// TwinCAT 3 PLC project Steamer
// ProgramVersion: 3.1.4026.25
// libraries:
//   Tc2_Standard, * (Beckhoff Automation GmbH)
//   Tc2_System, * (Beckhoff Automation GmbH)
//   Tc2_Utilities, * (Beckhoff Automation GmbH)
// project tree:
//   DUTs/Enumerations/ E_FaultId.TcDUT, E_HmiMessage.TcDUT (not stored), E_SystemState.TcDUT, E_WaterFillMode.TcDUT (not stored)
//   DUTs/Structures/ ST_Faults.TcDUT, ST_HmiCommand.TcDUT, ST_HmiSetpoints.TcDUT, ST_HmiStatus.TcDUT, ST_ProcessValues.TcDUT
//   GVLs/ GVL_HMI.TcGVL, GVL_IO.TcGVL, GVL_SysParameters.TcGVL
//   / PlcTask.TcTTO
//   POUs/ FB_FaultMonitor.TcPOU, FB_Hmi.TcPOU, FB_ProcessCalcs.TcPOU, FB_OutputHandler.TcPOU, FB_PressureControl.TcPOU, FB_Purge.TcPOU, FB_SpaFlush.TcPOU, FB_StateMachine.TcPOU, FB_WaterFill.TcPOU, MAIN.TcPOU
// real-time tasks:
//   TASK PlcTask: cycle T#10ms, priority 20, ADS port 350
// I/O:
//   DEVICE Device 1 (EtherCAT), AmsNetId 5.177.96.78.2.1
//     Term 1 (EK1200) [EK1200-7000 EtherCAT Power supply (1,5A E-Bus)]
//       Term 2 (EL1008) [EL1008 8Ch. Dig. Input 24V, 3ms]
//       Term 3 (EL2008) [EL2008 8Ch. Dig. Output 24V, 0.5A]
//       Term 4 (EL2008) [EL2008 8Ch. Dig. Output 24V, 0.5A]
//       Term 11 (EL3052) [EL3052 2Ch. Ana. Input 4-20mA]
//       Term 5 (EL3314) [EL3314 4Ch. Ana. Input Thermocouple (TC)]
//       Term 13 (EL6652-0010) [EL6652-0010 EtherNet/IP Adapter (Slave)]
//       Term 6 (EL9011) [EL9011 End Terminal]
// variable links:
//   Steamer/Steamer Instance <-> Device 1 (EtherCAT)/Term 1 (EK1200)/Term 11 (EL3052)
//     PlcTask Inputs/GVL_IO.aiPT1_UpstreamPressure <-> AI Standard Channel 1/Value
//     PlcTask Inputs/GVL_IO.aiPT2_DownstreamPressure <-> AI Standard Channel 2/Value
//   Steamer/Steamer Instance <-> Device 1 (EtherCAT)/Term 1 (EK1200)/Term 2 (EL1008)
//     PlcTask Inputs/GVL_IO.biLS1_WaterMidLevel <-> Channel 3/Input
//     PlcTask Inputs/GVL_IO.biLS2_WaterHighLevel <-> Channel 4/Input
//     PlcTask Inputs/GVL_IO.biLS3_WaterLowLevel <-> Channel 5/Input
//     PlcTask Inputs/GVL_IO.biTankFloodFault <-> Channel 2/Input
//   Steamer/Steamer Instance <-> Device 1 (EtherCAT)/Term 1 (EK1200)/Term 3 (EL2008)
//     PlcTask Outputs/GVL_IO.boH1_UpstreamHeater <-> Channel 5/Output
//     PlcTask Outputs/GVL_IO.boH2_SpaHeater <-> Channel 6/Output
//     PlcTask Outputs/GVL_IO.boH3_FlowmeterHeater <-> Channel 7/Output
//     PlcTask Outputs/GVL_IO.boH4_ExternalHeater <-> Channel 8/Output
//     PlcTask Outputs/GVL_IO.boSV1_DrainValve <-> Channel 1/Output
//     PlcTask Outputs/GVL_IO.boSV2_SpaValve <-> Channel 2/Output
//     PlcTask Outputs/GVL_IO.boSV3_DeliveryValve <-> Channel 3/Output
//     PlcTask Outputs/GVL_IO.boSV4_WaterInletValve <-> Channel 4/Output
//   Steamer/Steamer Instance <-> Device 1 (EtherCAT)/Term 1 (EK1200)/Term 5 (EL3314)
//     PlcTask Inputs/GVL_IO.aiTC1_SpaTemp <-> TC Inputs Channel 1/Value
//     PlcTask Inputs/GVL_IO.aiTC2_FlometerTemp <-> TC Inputs Channel 2/Value
//     PlcTask Inputs/GVL_IO.aiTC3_ExternalTemp <-> TC Inputs Channel 3/Value
//     PlcTask Inputs/GVL_IO.aiTC4_DeliveryTemp <-> TC Inputs Channel 4/Value

CONFIGURATION Steamer
    RESOURCE PLC ON TwinCAT3
        TASK PlcTask(INTERVAL := T#10ms, PRIORITY := 20);
        PROGRAM MAIN WITH PlcTask : MAIN;
    END_RESOURCE
END_CONFIGURATION

// ---- DUTs/Enumerations/E_FaultId.TcDUT
//=============================================================================
// E_FaultId
//-----------------------------------------------------------------------------
// Identifies WHICH fault tripped first. FB_FaultMonitor latches one of these
// on the transition from healthy to faulted and holds it until ResetAll().
//
// The numeric values are the legacy HMI message-table indices, so the existing
// message strings on the panel keep working without a translation layer.
// Where the legacy reused one index for several distinct causes, the causes
// are split into separate IDs here and the duplicated index is noted.
//=============================================================================
{attribute 'qualified_only'}
{attribute 'strict'}
{attribute 'to_string'}
TYPE E_FaultId :
(
    None                    := 0,

    // --- hardware / utilities -------------------------------------------
    PowerFault              := 1,
	CabinetFlood            := 2,
    PneumaticLow            := 3,

    // --- pressure -------------------------------------------------------
    UpstreamOverPress       := 11,
    DownstreamOverPress     := 12,
    DownstreamStartHigh     := 13,
    StartupDiffPressTimeout := 14,
    Pt1Hardware             := 15,
    Pt2Hardware             := 16,

    // Transducer cross-check failure. Legacy shared index 58 with the
    // timeout above; split so first-out can tell them apart. Point the HMI
    // message table at 58 if a distinct string is not wanted.
    StartupDiffPressXCheck  := 17,

    // --- water ----------------------------------------------------------
    WaterFill               := 21,
    WaterRegulation         := 22,
    WaterEmpty              := 23,
	WaterOverFill			:= 24,
    VesselPurgeTimeout      := 25,

    // --- temperature: over-limit ----------------------------------------
    SpaOverTemp             := 31,
    FlowMeterOverTemp       := 32,
    ExternalOverTemp        := 33,
    DownstreamOverTemp      := 34,

    // --- temperature: warm-up failures ----------------------------------
    SpaWarmupTimeout        := 41,
    FlowMeterWarmupTimeout  := 42,
    ExternalWarmupTimeout   := 43,
    DownstreamWarmupTimeout := 44,

    // Legacy reused index 76 for all three external-line faults. Split so
    // the operator can tell "TC not bonded to heater" from "line went cold".
    ExternalNoTempRise      := 51,
    ExternalLowAtReady      := 52,

    // --- flow -----------------------------------------------------------
    FlowRateError           := 61,

    // --- new in this system ---------------------------------------------
    HmiCommLoss             := 300
) INT;
END_TYPE

// ---- DUTs/Enumerations/E_SystemState.TcDUT
{attribute 'qualified_only'}
{attribute 'strict'}
{attribute 'to_string'}
TYPE E_SystemState :
(
    // --- Boot / idle ---------------------------------------------------
    InitController      := 0, 	// Controller Initialization (one-shot config, params, PID setup)
    SesOff              := 70,  // SES Off (idle / standby, waiting for SES ON command)

    // --- Startup sequence ----------------------------------------------
    CheckIfHot          := 10,  // Check if system was just running (hot restart shortcut)
    FillWater       	:= 20,  // SES Initialization - Fill Water
    PurgeVessel     	:= 30,  // SES Initialization - Purge Vessel
    SetDiffPressure 	:= 40,  // SES Initialization - Setting Differential Pressure
    InitMain       		:= 50,  // SES Initialization - Main (final checks before flow)

    // --- Run -------------------------------------------------------------
    SteamFlowing        := 60,  // Steam Flowing (normal production, PID flow control)

    // --- Service / abnormal ----------------------------------------------
    Maintenance         := 80,  // Maintenance mode (manual actuation, loopback)
    Fault               := 99   // Fault (latched; operator reset returns to InitController)
	
) INT;
END_TYPE

// ---- DUTs/Structures/ST_Faults.TcDUT
//=============================================================================
// ST_Faults
//-----------------------------------------------------------------------------
// One named BOOL per fault, replacing the legacy B1600.x / B1601.x / B1602.x
// bit-of-word addressing. Names taken from the element documentation table
// in the DS6 source. Legacy address noted per field for commissioning.
// pack_mode 1: each BOOL = 1 byte, so pyads can map this with a simple
// structure_def or read it as a byte array.
//=============================================================================
{attribute 'pack_mode' := '1'}
TYPE ST_Faults :
STRUCT
	// --- Legacy system faults --------------------------------------------
    bAnyFault					: BOOL;   	// High when any fault is active
    bPowerFault          		: BOOL;   	// Power fault input high
	bCabinetFlood        		: BOOL;   	// Cabinet flood fault
    bPneumaticLow        		: BOOL;   	// Pneumatic air pressure low
    bUpstreamOverPress   		: BOOL;   	// Upstream over pressure
    bDownstreamOverPress 		: BOOL;   	// Downstream over pressure
    bPt1HardwareFault      		: BOOL;   	// PT1 hardware fault
    bPt2HardwareFault      		: BOOL;   	// PT2 hardware fault
	bSpaOverTemp				: BOOL;		// SPA greater than max temp stpt
	bFlowmeterOverTemp			: BOOL;		// fm greater then max temp stpt
	bExtOverTemp				: BOOL;		// external temp greater than max stpt
	bDownstreamOverTemp			: BOOL;		// delivery temp greater than max stpt
	bSpaWarmupTimeout			: BOOL;		// spa temp below stpt after timeout
	bFlowmeterWarmupTimeout		: BOOL;		// fm temp below stpt after timeout
	bExtWarmupTimeout			: BOOL;		// external temp below stpt after timeout
	bDownstreamWarmupTimeout	: BOOL;		// ds temp below stpt after timeout
	bExtTempDecoupled			: BOOL;		// external temp disconnected from heater
	bExtTempLow					: BOOL;		// external temp low after steam ready
    bWaterEmpty          		: BOOL; 	// empty water level fault
	bWaterOverFill				: BOOL;		// water too full fault
	bWaterFillTimeout          	: BOOL; 	// water not full after timeout 
	bWaterDrainTimeout          : BOOL; 	// water not empty after timeout
	bWaterRegulationFault		: BOOL;		// water PID stuck on too long
	bPurgeTimeout				: BOOL;		// vessel purge incomplete after timeout
	bDownstreamStartOverPress	: BOOL;		// vessel not properly vented before restart
	bStartDpTimeout				: BOOL;		// diff pressure timeout before reaching stpt
	bStartDpHardwareFault		: BOOL;		// pressure outside of allowable variance
	bFlowFault					: BOOL;		// flow to dp ratio exceeds calibrated max

    // --- New-system faults ---------------------------------------
    bHmiCommLoss         : BOOL;   // (new) RPi heartbeat timeout
	
END_STRUCT
END_TYPE

// ---- DUTs/Structures/ST_HmiCommand.TcDUT
//=============================================================================
// ST_HmiCommand
//-----------------------------------------------------------------------------
// Direction: Pi -> PLC. Consume-on-read pattern:
//   * Pi writes TRUE to a command bit (pyads write_by_name).
//   * FB_Hmi latches it into its outputs for exactly one PLC cycle,
//     then writes FALSE back. The Pi never needs to clear anything.
//
//=============================================================================
{attribute 'pack_mode' := '1'}
TYPE ST_HmiCommand :
STRUCT
	// --- Heartbeat -------------------------------------------------------------
    nHmiHeartbeat   : UDINT;   // Pi increments each poll cycle; never reset

    // --- Run page buttons ---------------------------------------------------
    bSesOn          	: BOOL;    // start command
    bSesOff         	: BOOL;    // stop command 
	bSteamDeliveryOn	: BOOL;    // steam delivery enable
	bSteamDeliveryOff	: BOOL;    // steam delivery disable

    // --- Alarms page --------------------------------------------------------
    bFaultReset     	: BOOL;    // reset all faults
    bFaultAck       	: BOOL;    // acknowledge (silences banner, faults stay listed)

    // --- Maintenance page ---------------------------------------------------
    bEnterMaint     	: BOOL;    				// request Maintenance state
    bExitMaint      	: BOOL;    				// leave Maintenance 
    aValveCmd      		: ARRAY[1..4] OF BOOL;  // SV1 drain, SV2 main, SV3 process, SV4 water
    bDrainMode      	: BOOL;    				// drain mode
	bDpControlOn   		: BOOL;    				// suspend diff pressure control
    bDpControlOff   	: BOOL;    				// suspend diff pressure control
	bTempControlOn	 	: BOOL;    				// suspend purifier temp control
    bTempControlOff 	: BOOL;    				// suspend purifier temp control
    bExtHeaterOn		: BOOL;    				// external heater enable
	bExtHeaterOff		: BOOL;					// extermal heater disable	
	bAutofillOn			: BOOL;					// toggle autofill enable when running
	bAutofillOff		: BOOL;					// toggle autofill off

    // --- Config page --------------------------------------------------------
    bApplySetpoints : BOOL;    // pulse: validate + apply stSetpointRequest

END_STRUCT
END_TYPE

// ---- DUTs/Structures/ST_HmiSetpoints.TcDUT
//=============================================================================
// ST_HmiSetpoints
//-----------------------------------------------------------------------------
// Direction: Pi -> PLC (request) and PLC -> Pi (applied echo in ST_HmiStatus).
// Pi writes the whole struct, then pulses stCommand.bApplySetpoints.
// FB_Hmi clamps each value to ST_SetpointLimits before applying, and the
// clamped result is echoed in ST_HmiStatus.rSet*Applied so the UI always
// shows the truth, not the request.
//=============================================================================
{attribute 'pack_mode' := '1'}
TYPE ST_HmiSetpoints :
STRUCT
	bSetPurgeOnStartup	: BOOL := FALSE;	// 
	rSetFlow       		: REAL;  			// requested flow setpoint      [SLM]
    //rSetDsPressure 		: REAL; 			// downstream pressure setpoint [Torr]
	rSetElevation		: REAL;				// meters above seal level [MASL] 
	bSetSize25L			: BOOL;				// set size to 25L, FALSE = 50L
	sSetEipAddress		: STRING(15);		// string to represent EthernetIP address
END_STRUCT
END_TYPE

// ---- DUTs/Structures/ST_HmiStatus.TcDUT
//=============================================================================
// ST_HmiStatus
//-----------------------------------------------------------------------------
// EVERYTHING the RPi HMI displays, packed into ONE struct so pyads can
// refresh the whole UI with a single read:
//     plc.read_by_name('GVL_HMI.stStatus', structure_def=ST_HMI_STATUS)
//
// Direction: PLC -> Pi only. The Pi must never write this struct.
// pack_mode 1: byte-aligned, no padding — pyads structure_def matches 1:1.
//=============================================================================
{attribute 'pack_mode' := '1'}
TYPE ST_HmiStatus :
STRUCT
    // --- Liveness / handshake -------------------------------------------
    nPlcHeartbeat    	: UDINT;             	// increments every PLC cycle group; Pi checks it changes
    nHmiHeartbeatEcho 	: UDINT;           		// last heartbeat value received from Pi (debug aid)
    bHmiOnline      	: BOOL;              	// PLC's view: Pi heartbeat is alive

    // --- System state ----------------------------------------------------
    eState          	: E_SystemState;     	// current state (INT under the hood)
    sStateName      	: STRING(31);        	// human-readable, e.g. 'SteamFlowing' (state pill)
    bReady          	: BOOL;              	// green Ready dot (temps in band, no faults)
    bAlarmActive    	: BOOL;              	// red Alarm dot (any fault bit set)
    nActiveFaults   	: UINT;              	// count of active fault bits (Alarms page stat card)

    // --- Process data ------------------------------------------------------
    stProcess       	: ST_ProcessValues;  	// pressures, temps, flow, water level
	bFillComplete		: BOOL;					// water fill complete
	rFlowPercent    	: REAL;              	// rFlowActual / rFlowRated * 100 (bar graph)
	
	// --- Faults -------------------------------------------------------------
	stFaults			: ST_Faults;			// process faults
	aActiveFaults		: ARRAY[1..2, 1..5] OF STRING(30);

    // --- PID loop outputs [0..100 %] (Run page bars) ------------------------
    arPidOutput     	: ARRAY[1..6] OF REAL;  // 1 dP, 2 SPA temp, 3 heater, 4 water, 5 FM temp, 6 spare

    // --- Setpoint echo (what the PLC actually accepted after clamping) ------
    rSetFlowApplied     : REAL;          		// SL
    rSetDsPressApplied  : REAL;          		// Torr
    rSetSpaTempApplied  : REAL;          		// degC

    // --- Maintenance feedback (Maintenance page) ----------------------------
    arValveState        : ARRAY[1..4] OF BOOL;  // SV1 drain, SV2 main, SV3 process, SV4 water
    bLoopbackOn         : BOOL;          		// legacy C31
    bDrainModeOn        : BOOL;

    // --- System info --------------------------------------------------------
    sPlcVersion     	: STRING(31);        	// version of the PLC program
    sHmiVersion     	: STRING(31);        	// echoed from Pi at startup, shown for record
    nUptimeSeconds  	: UDINT;

END_STRUCT
END_TYPE

// ---- DUTs/Structures/ST_ProcessValues.TcDUT
//=============================================================================
// ST_ProcessValues
//-----------------------------------------------------------------------------
// Live process data in ENGINEERING UNITS (Torr, degC, SLM).
// Populated by FB_FlowCalc / analog input scaling, consumed by FB_Hmi,
// FB_FaultMonitor and FB_PressureControl.
// pack_mode 1 so pyads structure_def offsets are byte-exact.
//=============================================================================
{attribute 'pack_mode' := '1'}
TYPE ST_ProcessValues :
STRUCT
    // --- Pressures [Torr] -------------------------------- 
    rPt1Upstream    	: REAL;    			// PT-1 upstream pressure    
    rPt2Downstream  	: REAL;    			// PT-2 downstream pressure  
    //rPt3AtmRef      	: REAL;    			// PT-3 atmospheric reference
    rDiffPressure   	: REAL;    			// PT-1 - PT-2 differential
	rDiffPressureOffset	: REAL;				// pt1-pt2 differential when equalized
	rAtmPressure		: REAL := 760;		// atmospheric pressure - computed

    // --- Temperatures [degC] ------------------------------
    rTc1Spa         	: REAL;    	// TC1 SPA temperature
    rTc2FlowMeter   	: REAL;    	// TC2 flow meter temperature
    rTc3External    	: REAL;    	// TC3 external heater temperature
    rTc4Delivery    	: REAL;    	// TC4 delivery line temperature

    // --- Flow [SLM] ---------------------------------------
    rFlowActual     	: REAL;    			// F3 calculated steam flow     
    rFlowSetpoint   	: REAL;    			// active flow setpoint         
    rFlowRated      	: REAL := 25.0;    	// rated max flow    
	rFlowRatio			: REAL;				// FL_TO_DP23 = F3 / DP23 --> units: SLM per Torr  
	rCondensateFlow		: REAL;				// flow through the small (drain/condensate) orifice         

    // --- Discrete process status --------------------------
    bWaterHigh			: BOOL;		// water at high limit --> high limit switch on
	bWaterFull      	: BOOL;    	// full water level --> center limit switch on, high off
    bWaterLow       	: BOOL;    	// low water level --> low limit switch on, center/high off
    bWaterEmpty     	: BOOL;    	// empty water level --> low limit switch off    
	bPowerFaultSensor 	: BOOL;		// power fault sensor
	bCabinetFloodSensor	: BOOL;		// cabinet flood sensor
	
END_STRUCT
END_TYPE

// ---- GVLs/GVL_HMI.TcGVL
//=============================================================================
// GVL_HMI
//-----------------------------------------------------------------------------
// The ONLY variables the RPi/pyads client touches. Three symbols, three jobs:
//
//   GVL_HMI.stStatus           PLC -> Pi   read-only  (one bulk read per poll)
//   GVL_HMI.stCommand          Pi -> PLC   buttons + heartbeat
//   GVL_HMI.stSetpointRequest  Pi -> PLC   config values, applied via
//                                          stCommand.bApplySetpoints
//
// Everything else in the PLC is off-limits to the HMI by convention.
// If the HMI needs a new value, add it to ST_HmiStatus — never let the
// Pi read internal FB state directly, or the interface contract rots.
//
// pyads access, e.g.:
//   plc = pyads.Connection('5.x.x.x.1.1', 851)
//   status = plc.read_by_name('GVL_HMI.stStatus', structure_def=HMI_STATUS_DEF)
//   plc.write_by_name('GVL_HMI.stCommand.bSesOn', True)
//=============================================================================
{attribute 'qualified_only'}
VAR_GLOBAL
    stHmiStatus         : ST_HmiStatus;      // PLC -> Pi
    stHmiCommand        : ST_HmiCommand;     // Pi -> PLC (FB_Hmi consumes+clears pulses)
END_VAR

VAR_GLOBAL PERSISTENT
	stHmiSetpoints 		: ST_HmiSetpoints;   // Pi -> PLC (applied on bApplySetpoints)
END_VAR

VAR_GLOBAL CONSTANT
    // Pi poll rate is expected >= 1 Hz; comm loss declared after this timeout
    T_HMI_HEARTBEAT_TIMEOUT : TIME := T#5S;
    S_PLC_VERSION           : STRING(31) := 'V 0.x';
END_VAR

// ---- GVLs/GVL_IO.TcGVL
{attribute 'qualified_only'}
VAR_GLOBAL
	
	// binary inputs
	//biPowerFault				AT %I* : BOOL;
	biTankFloodFault			AT %I* : BOOL;
	biLS1_WaterMidLevel			AT %I* : BOOL;
	biLS2_WaterHighLevel		AT %I* : BOOL;
	biLS3_WaterLowLevel			AT %I* : BOOL;
	//biPS1_						AT %I* : BOOL;
	                        	
	// binary outputs       	
	boSV1_DrainValve			AT %Q* : BOOL;
	boSV2_SpaValve				AT %Q* : BOOL;
	boSV3_DeliveryValve			AT %Q* : BOOL;
	boSV4_WaterInletValve		AT %Q* : BOOL;
	boH1_UpstreamHeater			AT %Q* : BOOL;
	boH2_SpaHeater				AT %Q* : BOOL;
	boH3_FlowmeterHeater		AT %Q* : BOOL;
	boH4_ExternalHeater			AT %Q* : BOOL;
	//boLED1_ReadyLight			AT %Q* : BOOL;
	//boLED2_AlarmLight			AT %Q* : BOOL;
	
	// analog inputs
	aiPT1_UpstreamPressure		AT %I* : INT;
	aiPT2_DownstreamPressure 	AT %I* : INT;
	aiTC1_SpaTemp				AT %I* : INT;
	aiTC2_FlometerTemp			AT %I* : INT;
	aiTC3_ExternalTemp			AT %I* : INT;
	aiTC4_DeliveryTemp			AT %I* : INT;	
	
END_VAR

// ---- GVLs/GVL_SysParameters.TcGVL
   {attribute 'qualified_only'}
// ------------------------- persisent vars -----------------------------------
VAR_GLOBAL
	
	// SV2 pressure relief and closing delay
		rUpstreamPressureReleived 	: REAL := 800;	// 800 Torr
		tSv2CloseDelay 				: TIME := T#5S;
	
	// --- State Machine ------------------------------------------------------
	
	// CheckIfHot state
		rSpaWarmMinimumTemp : REAL := 30.0;		// 30 degC --> TODO: check if this value makes sense
		rHotRestartFlowPct 	: REAL := 10.0;    	// current flow is over x% of rated flow	


	// SteamFlowing State
		rFlowDeadbandPct 	: REAL := 0.10;		// deadband target of steam flow as %

	// ------------------------------------------------------------------------	
	// --- Function Blocks ----------------------------------------------------

	// FB_WaterFill
		tDebounceTimer 			: TIME := T#2S;
		tStartupFillTimeout		: TIME := T#15M;
		tFillConfirmDelay		: TIME := T#5S;
		tAutoFillTimeout		: TIME := T#1M;
		tStartupFillDelay		: TIME := T#10s;
		tAutoFillDelay			: TIME := T#4S;	
		tAutofillPidSample		: TIME := T#1s;
	
	// FB_Purge
		rAtmosphericPressure	: REAL := 760; 							// [torr] default, calc'd in FB_Purge 
		rPurgeTargetPressure	: REAL := rAtmosphericPressure + 50; 	// [torr]
		rPurgeBand				: REAL := 20; 							// [torr]
		tDrainOpen				: TIME := T#1S;
		tEquilibrate			: TIME := T#5S;
		tPurgeTimeout			: TIME := T#15M;
	
	// FB_PressureControl
		tPidSampleTime			: TIME := T#50MS;
		
		// --- loop 1: boiler / upstream pressure -> H1 ---------------------------
		rPid1_Kp				: REAL := 25.0;		// [%/Torr]
		rPid1_Ti				: REAL := 20.0;		// [s]  legacy = K200 -> 20.0
		rPid1_Td				: REAL := 0.0;		// [s]  legacy = K0
		tPid1PwmPeriod			: TIME := T#2S;		// legacy = K200 (0.01 s units)
		tPid1PwmPeriodSlow		: TIME := T#4S;		// legacy = K400, purge / pre-flush
		tPid1MaxOnTime			: TIME := T#2S;		// legacy = 200 counts. Fixed, so the slow period caps at 50 %.
		rIniDeltaPressure		: REAL := 100.0;	// [Torr] pre-flush SP above PT3
		rPspGainOffset			: REAL := 0.0;		// [Torr] Never initialised in legacy
		tSpRampInterval			: TIME := T#500MS;	// legacy = K5 (0.1 s units)
		rSpRampStep				: REAL := 1.0;		// [Torr] per interval -> 2 Torr/s
		rSpaTempSp				: REAL := 75;		// temp setpoint
	 
		// --- loop 2: SPA / purifier temperature -> H2 ---------------------------
		rPid2_Kp				: REAL := 20.0;		// [%/degC]
		rPid2_Ti				: REAL := 15.0;		// [s]  legacy = K150
		rPid2_Td				: REAL := 0.0;		// [s]  legacy = K50. Consider 0 until loop is characterised
		tPid2PwmPeriod			: TIME := T#100MS;	// legacy = K10
	 
		// --- loop 3: flow meter temperature -> H3 -------------------------------
		rPid3_Kp				: REAL := 2000.0;	// [%/degC]
		rPid3_Ti				: REAL := 15.0;		// [s]
		rPid3_Td				: REAL := 5.0;		// [s]
		tPid5PwmPeriod			: TIME := T#100MS;	// legacy V1530 = K10
		rFlowMeterTempSp		: REAL := 120.0;	// [degC] legacy = K1200
		rDeliveryTempCutout		: REAL := 140.0;	// [degC] legacy = K1400, TC4 at or above this inhibits H3.
		rFlowMin				: REAL := 2.5;
		rFlowMax				: REAL := 25;
	 
		// --- loop 4: external line heater -> H4 (bang-bang) ---------------------
		rExtHeaterTempSp		: REAL := 120.0;	// [degC] legacy V1521 = K1200
		
	// FB_FaultMonitor
		rUpstreamMaxPressure	: REAL := 1530; 	// torr
		rDownstreamMaxPressure	: REAL := 1250;		// torr
		rPtMininum				: REAL := 50;		// minimum reading --> hardware fault
		rMaxTemp				: REAL := 150.0;	// [degC]
 		rWarmupTemp				: REAL := 30.0;		// degC, minimum temp during warmup
		rExtTempMinRise			: REAL := 5.0;		// minimum temp to rise without triggering ext fault
		rExtMinReadyTemp		: REAL := 95.0;		// external heater low limit when steam ready
		rDsHighStartPressure	: REAL := 1500.0;	// max starting pressure for downstream sensor
		rP3AbsMax				: REAL := 785.0;	// max atmospheric pressure 
		rP3AbsMin				: REAL := 575.0;	// min atmospheric pressure
		rPtMaxVariance			: REAL := 10.0;		// 
		rMaxFlowDpRatio			: REAL := 0.25;		// rated_flow(×10 SLM) × 0.001 = 250 × 0.001 = 0.25 SLM/Torr
	
	
END_VAR

// ---- POUs/MAIN.TcPOU
PROGRAM MAIN
VAR
	// HMI Variables
	HMI_bRun 	: BOOL;
	HMI_nPT1	: INT;
	
	// state machine
	eSystemState		: E_SystemState;

	// function blocks
	fbProcessCalcs		: FB_ProcessCalcs;
	fbFaultMonitor 		: FB_FaultMonitor;
	fbHmi 				: FB_Hmi;
	fbPressureControl 	: FB_PressureControl;
	fbPurge 			: FB_Purge;
	fbSpaFlush			: FB_SpaFlush;
	fbStateMachine 		: FB_StateMachine;
	fbWaterFill 		: FB_WaterFill;
	fbOutputHandler		: FB_OutputHandler;
	
	// fbWaterFill
	reqSV4_FillVavle			: BOOL;
	bLS1_WaterCenter_Filtered	: BOOL;
	bLS3_WaterEmpty_Filtered	: BOOL;
	
	// fbPurge
	reqSV1_DrainValve			: BOOL;
	
	// fbPresureControl
	reqH1_Upstream				: BOOL;
	
END_VAR

//========================= FB CALLS =====================================

// SCALE INPUTS
fbProcessCalcs(eState := fbStateMachine.eState);

// FAULT CHECK
fbFaultMonitor(
	stProcess := fbProcessCalcs.stProcessValues,
	eState := fbStateMachine.eState,
	bPurgeActive := fbStateMachine.bPurgeEnable,
	bWaterFillActive := (fbWaterFill.eMode = E_WaterFillMode.RunningAutofill) 
						 OR (fbWaterFill.eMode = E_WaterFillMode.StartupFill),
	bDiffPressActive := fbStateMachine.bControlEnable,
	bDiffPressReached := fbPressureControl.bDiffPressReached,
	bTempControlActive := fbStateMachine.bControlEnable,
	bColdStart := fbStateMachine.bColdStart,
	bReadyReached := fbStateMachine.bReady,
	bSteamFlowing := fbStateMachine.bDeliveryEnable,
	bWaterEmptyFiltered := fbWaterFill.bEmptyFiltered,
	bWaterCenterFiltered := fbWaterFill.bCenterFiltered,
	bExternalHeaterOff := NOT fbStateMachine.bExtHeaterEnable,
	bHmiHeartbeatOk := NOT fbHmi.bHmiCommLoss
	);
	
// Latch fault -> force state machine into Fault (only auto-clears via reset).
IF fbFaultMonitor.bAnyLatchingFault THEN
    fbStateMachine.RequestFault();
END_IF

//========================= HMI (publish + consume) =======================
// Run BEFORE the state machine so command pulses are latched this cycle.
// FB_Hmi publishes GVL_HMI.stStatus and clears consumed command bits.
fbHmi(
	eState      				:= fbStateMachine.eState,
    stProcess   				:= fbProcessCalcs.stProcessValues,
	stFaults					:= fbFaultMonitor.stFaults,
	aActiveFaults				:= fbFaultMonitor.aActiveFaults,
	bReady 						:= fbStateMachine.bReady
);
	  
// Consume the one-cycle HMI command pulses
IF fbHmi.bCmdSesOn THEN fbStateMachine.RequestStart(); END_IF
IF fbHmi.bCmdSesOff THEN fbStateMachine.RequestStop(); END_IF
IF fbHmi.bCmdDeliveryOn THEN fbStateMachine.RequestDelivery(TRUE); END_IF
IF fbHmi.bCmdDeliveryOff THEN fbStateMachine.RequestDelivery(FALSE); END_IF
IF fbHmi.bCmdFaultReset THEN fbFaultMonitor.ResetAll(); fbStateMachine.RequestFaultReset(); END_IF;
// IF fbHmi.bCmdFaultAck THEN ...
IF fbHmi.bCmdEnterMaint THEN fbStateMachine.RequestMaintenance(); END_IF
IF fbHmi.bCmdExitMaint THEN fbStateMachine.RequestExitMaint(); END_IF
IF fbHmi.bCmdExtHeaterOn THEN fbStateMachine.RequestExtHeater(TRUE); END_IF
IF fbHmi.bCmdExtHeaterOff THEN fbStateMachine.RequestExtHeater(FALSE); END_IF
IF fbHmi.bCmdAutofillOn THEN fbStateMachine.RequestAutofill(TRUE); END_IF
IF fbHmi.bCmdAutofillOff THEN fbStateMachine.RequestAutofill(FALSE); END_IF
IF fbHmi.bCmdDpLoopOn THEN fbStateMachine.RequestDpLoop(TRUE); END_IF
IF fbHmi.bCmdDpLoopOff THEN fbStateMachine.RequestDpLoop(FALSE); END_IF
IF fbHmi.bCmdTempLoopOn THEN fbStateMachine.RequestTempLoop(TRUE); END_IF
IF fbHmi.bCmdTempLoopOff THEN fbStateMachine.RequestTempLoop(FALSE); END_IF
IF fbHmi.bCmdApplySetpoints THEN 
	IF GVL_HMI.stHmiSetpoints.rSetFlow < GVL_SysParameters.rFlowMin THEN GVL_HMI.stHmiSetpoints.rSetFlow := GVL_SysParameters.rFlowMin; END_IF
	IF GVL_HMI.stHmiSetpoints.rSetFlow > GVL_SysParameters.rFlowMax THEN GVL_HMI.stHmiSetpoints.rSetFlow := GVL_SysParameters.rFlowMax; END_IF
END_IF

//========================= STATE MACHINE =================================

fbStateMachine(
	stFaults := fbFaultMonitor.stFaults,
	stHmiSetpoints := GVL_HMI.stHmiSetpoints,
	stProcessValues := fbProcessCalcs.stProcessValues,
	bFillComplete := fbWaterFill.bFillComplete,
	bPurgeComplete := fbPurge.bPurgeComplete,
	bSpaFlushed := fbSpaFlush.bSpaFlushed,
	bDpReached := fbPressureControl.bDiffPressReached,
	eState => eSystemState
);
				
//========================= SUBROUTINES =================================
// Subroutines only run only when the state machine enables them. In Maintenance,
// the enable flags follow the HMI control-loop override toggles.

fbWaterFill(
	eMode := fbStateMachine.eWaterFillMode,
	rSteamFlow := fbProcessCalcs.stProcessValues.rFlowActual,
	bCenterSwitch := GVL_IO.biLS1_WaterMidLevel,
	bEmptySwitch := GVL_IO.biLS3_WaterLowLevel,
	bAutofillEnable := fbStateMachine.bAutofillEnable,
	bFillComplete => GVL_HMI.stHmiStatus.bFillComplete,
	bCenterFiltered => GVL_HMI.stHmiStatus.stProcess.bWaterFull,
	bEmptyFiltered => GVL_HMI.stHmiStatus.stProcess.bWaterEmpty
);

fbPurge(
	bEnable :=fbStateMachine.bPurgeEnable,
	rUpstreamPress := fbProcessCalcs.stProcessValues.rPt1Upstream,
	bEmptyFiltered := fbWaterFill.bEmptyFiltered,
	bPurgeTimeout => GVL_HMI.stHmiStatus.stFaults.bPurgeTimeout
);
		

fbSpaFlush(
	bEnable := fbStateMachine.bSpaFlushEnable,
	bReset := fbStateMachine.bSpaFlushReset,
	rUpstreamPress := fbProcessCalcs.stProcessValues.rPt1Upstream,
	rAtmPressure := fbProcessCalcs.stProcessValues.rAtmPressure
);
	
fbPressureControl(
	bEnable := fbStateMachine.bControlEnable,          
	eState := fbStateMachine.eState,        
	bDpControlOff := NOT fbStateMachine.bDpLoopEnable,
	bTempControlOff := NOT fbStateMachine.bTempLoopEnable,
	bExtHeaterEnable := fbStateMachine.bExtHeaterEnable,
	stProcess := fbProcessCalcs.stProcessValues,
	stSetpoints := GVL_HMI.stHmiSetpoints ,
	bFlushed := fbSpaFlush.bSpaFlushed,
	bSpaPressurized := fbSpaFlush.bSpaPressurized
);



//========================= OUTPUT HANDLER ====================================
fbOutputHandler(
	eState := fbStateMachine.eState,
	bWaterFillValve := fbWaterFill.qFillValve,
	bPurgeValve := fbPurge.qDrainValve,
	bDeliveryPermit := fbStateMachine.bDeliveryEnable,
	bH1Upstream := fbPressureControl.qH1_UpstreamHeater,
	bH2Purifier := fbPressureControl.qH2_SpaHeater,
	bFmHeater := fbPressureControl.qH3_FlowmeterHeater,
	bExtHeater := fbPressureControl.qH4_ExternalHeater,
	arValveOverride := GVL_HMI.stHmiCommand.aValveCmd,
	stProcess := fbProcessCalcs.stProcessValues
);

END_PROGRAM

// ---- POUs/FB_ProcessCalcs.TcPOU
FUNCTION_BLOCK FB_ProcessCalcs
VAR_INPUT
	eState				: E_SystemState;
END_VAR
VAR_OUTPUT
    stProcessValues 	: ST_ProcessValues;   		// this FB is the only writer
END_VAR

VAR
	// pressure calculations
	rCurrentMeasRange	: REAL := 32767; 		// 16bit signed INT --> 0-32767 is positive range
	rSensorPressRange	: REAL := 1551.45;		// 0-30psia --> 0-1551.45torr
	
	// flow calculations
	rDp12 				: REAL;
	rDp23				: REAL;
	rFlowActual			: REAL;
	rOrificeA1_25		: REAL := 0.05946087;	// main orifice coefficient
	rOrificeA1_50		: REAL := 0.09;			// main orifice coefficient
	rOrificeA2			: REAL := 0.001057082;	// condensate/drain path coefficient
	rOrificeA3			: REAL := 0.01;			// SPA path coefficient
	rOrificeB1			: REAL := 0.0;			// main orifice offset
	rOrificeB2			: REAL := 0.0;	 		// condensate offset
	rOrificeB3			: REAL := 40; 			// torr offset
	
END_VAR

// temperature calculations
stProcessValues.rTc1Spa := TO_REAL(GVL_IO.aiTC1_SpaTemp)/10;
stProcessValues.rTc2FlowMeter := TO_REAL(GVL_IO.aiTC2_FlometerTemp)/10;
stProcessValues.rTc3External := TO_REAL(GVL_IO.aiTC3_ExternalTemp)/10;
stProcessValues.rTc4Delivery := TO_REAL(GVL_IO.aiTC4_DeliveryTemp)/10;

// pressure calculations
stProcessValues.rPt1Upstream := TO_REAL(GVL_IO.aiPT1_UpstreamPressure)/rCurrentMeasRange * rSensorPressRange;
stProcessValues.rPt1Upstream := stProcessValues.rPt1Upstream - stProcessValues.rDiffPressureOffset;
stProcessValues.rPt2Downstream := TO_REAL(GVL_IO.aiPT2_DownstreamPressure)/rCurrentMeasRange * rSensorPressRange;
stProcessValues.rDiffPressure := stProcessValues.rPt1Upstream - stProcessValues.rPt2Downstream;

IF eState = E_SystemState.FillWater AND stProcessValues.rTc1Spa < 30 AND stProcessValues.rTc2FlowMeter < 30 THEN
	stProcessValues.rAtmPressure := stProcessValues.rPt2Downstream;
	stProcessValues.rDiffPressureOffset := (TO_REAL(GVL_IO.aiPT1_UpstreamPressure)/rCurrentMeasRange * rSensorPressRange) - 
										   (TO_REAL(GVL_IO.aiPT2_DownstreamPressure)/rCurrentMeasRange * rSensorPressRange);
END_IF

// flow calculations
stProcessValues.rFlowSetpoint := GVL_HMI.stHmiSetpoints.rSetFlow;

rDp23 := stProcessValues.rPt2Downstream - stProcessValues.rAtmPressure;
IF rDp23 > 0.0 THEN
	stProcessValues.rFlowRatio := stProcessValues.rFlowActual / rDp23;
    stProcessValues.rCondensateFlow :=
        MAX(rOrificeA2 * SQRT(rDp23 * stProcessValues.rAtmPressure) - rOrificeB2, 0.0);
ELSE
	stProcessValues.rFlowRatio := 0.0;      
    stProcessValues.rCondensateFlow := 0.0;
END_IF

// actual delivered flow 
IF stProcessValues.rPt1Upstream > stProcessValues.rPt2Downstream THEN
	IF gvl_HMi.stHmiSetpoints.bSetSize25L THEN
		rFlowActual := rOrificeA1_25 * SQRT(stProcessValues.rDiffPressure * stProcessValues.rPt2Downstream)
			   - rOrificeB1 - stProcessValues.rCondensateFlow;
	ELSE
		rFlowActual := rOrificeA1_50 * SQRT(stProcessValues.rDiffPressure * stProcessValues.rPt2Downstream)
			   - rOrificeB1 - stProcessValues.rCondensateFlow;
	END_IF
    stProcessValues.rFlowActual := MAX(rFlowActual, 0.0);
ELSE
    stProcessValues.rFlowActual := 0.0;
END_IF

// discrete signals
stProcessValues.bWaterHigh := GVL_IO.biLS2_WaterHighLevel;
stProcessValues.bWaterFull := GVL_IO.biLS1_WaterMidLevel AND NOT GVL_IO.biLS2_WaterHighLevel;
stProcessValues.bWaterLow := GVL_IO.biLS3_WaterLowLevel AND NOT GVL_IO.biLS1_WaterMidLevel;
stProcessValues.bWaterEmpty := NOT GVL_IO.biLS3_WaterLowLevel;
stProcessValues.bCabinetFloodSensor  := GVL_IO.biTankFloodFault;

GVL_HMI.stHmiStatus.stProcess := stProcessValues;

END_FUNCTION_BLOCK

// ---- POUs/FB_FaultMonitor.TcPOU
FUNCTION_BLOCK FB_FaultMonitor
VAR_INPUT
    // --- scaled process values ------------------------------------------
    stProcess           : ST_ProcessValues;

    // --- sequence context (drives scope gating) -------------------------
    eState              : E_SystemState;
	eFaultId			: E_FaultId;
    bPurgeActive        : BOOL;   // TRUE while the purge sequence runs
    bWaterFillActive    : BOOL;   // TRUE while a fill is being commanded
    //bWaterFillRequest   : BOOL;   // for water regulation fault --> currently off
    bDiffPressActive    : BOOL;   // TRUE while differential pressure is being established
    bDiffPressReached   : BOOL;   // upstream pressure reached target setpoint
    bTempControlActive  : BOOL;   // TRUE while the heater loops are enabled
    bColdStart          : BOOL;   // one-shot: cold start, arm the temperature-rise check
    bReadyReached       : BOOL;   // steam-ready has been achieved at least once
    bSteamFlowing       : BOOL;   // production state

    // --- filtered level switches ----------------------------------------
    bWaterEmptyFiltered : BOOL;   // filtered lower limit switch: TRUE = vessel empty
    bWaterCenterFiltered: BOOL;   // filtered centre limit switch: TRUE = water present

    // --- configuration ---------------------------------------------------
    bExternalHeaterOff  : BOOL;   // external heater not installed / disabled
    bHmiHeartbeatOk     : BOOL;   // RPi heartbeat healthy
END_VAR
VAR_OUTPUT
    stFaults            : ST_Faults;
    bAnyLatchingFault   : BOOL;   		// mirrors stFaults.bAnyFault, for MAIN
    aActiveFaults		: ARRAY[1..2, 1..5] OF STRING(30);
END_VAR
VAR
    // --- reset-window suppression ----------------------------------------
    bSensorHwInhibit    : BOOL;

    // --- filter timers: periodic checks -----------------------------------
    tonPneumaticLow     : TON;
	tPneumaticFilter	: TIME := T#6S;
    tonUpstreamHigh     : TON;
    tonDownstreamHigh   : TON;
    tonPt1Bad           : TON;
    tonPt2Bad           : TON;
    tonSpaOverTemp      : TON;
    tonFmOverTemp       : TON;
    tonExtOverTemp      : TON;
    tonDsOverTemp       : TON;

	tGeneral_250ms		: TIME := T#250MS;
	tGeneral_10s		: TIME := T#10S;
	
    // --- sequence watchdogs ------------------------------------------------
    tonWarmup           : TON;
	tWarmup				: TIME := T#300S;
    tonPurge            : TON;
    tonDiffPress        : TON;
	tDiffPressTimeout	: TIME := T#20M;
    tonWaterFill        : TON;
    tonWaterReg         : TON;
    tonWaterEmpty       : TON;
	tonWaterOverfill    : TON;
	
	tWater_15m			: TIME := T#15M;
	tFullDelay			: TIME := T#5S;

    // --- external-line temperature checks ---------------------------------
    tonExtWarmupWindow  : TON;   			// fixed window for the temperature-rise test
	tExtRiseTimeout		: TIME := T#120S;	// delay to allow ext temp rise on cold start
    tonExtLowAtReady    : TON;
    rExtTempAtStart     : REAL;  			// external temperature captured at cold start
    bExtRiseArmed       : BOOL;
    bExtRiseTested      : BOOL;

    // --- flow ratio check --------------------------------------------------
    tonFlowRatio        : TON;
	tFlowRatioFilter	: TIME := T#1M;

    // --- edge detection ----------------------------------------------------
    rtColdStart         : R_TRIG;
    bAnyFaultPrev       : BOOL;
END_VAR

//--- Power fault. No filter: this is a hard utility loss. -------------------
IF stProcess.bPowerFaultSensor THEN
    stFaults.bPowerFault := TRUE;
    _Report(E_FaultId.PowerFault);
END_IF

//--- Cabinet flood. Sensor is normally closed, so LOSS of the input is the
//    alarm condition. A severed cable trips the fault, which is the intent.
IF NOT stProcess.bCabinetFloodSensor THEN
    stFaults.bCabinetFlood := TRUE;
    _Report(E_FaultId.CabinetFlood);
END_IF

//--- Pneumatic supply low. Also normally closed: open contact = low air.
//    Filtered because supply pressure dips briefly on every valve actuation.
(* tonPneumaticLow(IN := NOT stProcess.bPneumaticPressureSwitch,
                PT := tPneumaticFilter);   // 6.0 s
IF tonPneumaticLow.Q THEN
    stFaults.bPneumaticLow := TRUE;
    _Report(E_FaultId.PneumaticLow);
END_IF *)

//--- Upstream over pressure. Short filter rejects transducer noise while
//    still tripping fast enough to matter on a real overpressure.
tonUpstreamHigh(IN := stProcess.rPt1Upstream > GVL_SysParameters.rUpstreamMaxPressure,
                PT := tGeneral_250ms);    // 250 ms
IF tonUpstreamHigh.Q THEN
    stFaults.bUpstreamOverPress := TRUE;
    _Report(E_FaultId.UpstreamOverPress);
END_IF

//--- Downstream over pressure. ---------------------------------------------
tonDownstreamHigh(IN := stProcess.rPt2Downstream > GVL_SysParameters.rDownstreamMaxPressure,
                  PT := tGeneral_250ms);
IF tonDownstreamHigh.Q THEN
    stFaults.bDownstreamOverPress := TRUE;
    _Report(E_FaultId.DownstreamOverPress);
END_IF

//--- Transducer health. A reading below the minimum credible pressure means
//    the transducer is disconnected or its loop supply is dead, not that the
//    vessel is genuinely at that pressure. Suppressed during the reset window
//    so a dead transducer does not deadlock the operator.
bSensorHwInhibit := (eState = E_SystemState.Fault);

tonPt1Bad(IN := (stProcess.rPt1Upstream < GVL_SysParameters.rPtMininum) AND NOT bSensorHwInhibit,
          PT := tGeneral_250ms);
IF tonPt1Bad.Q THEN
    stFaults.bPt1HardwareFault := TRUE;
    _Report(E_FaultId.Pt1Hardware);
END_IF

tonPt2Bad(IN := (stProcess.rPt2Downstream < GVL_SysParameters.rPtMininum) AND NOT bSensorHwInhibit,
          PT := tGeneral_250ms);
IF tonPt2Bad.Q THEN
    stFaults.bPt2HardwareFault := TRUE;
    _Report(E_FaultId.Pt2Hardware);
END_IF

//--- Over-temperature, all four channels against the shared maximum.
//    NOTE: the legacy latched NO bit for any of these four - it only pushed a
//    message and jumped. Named latches added so bAnyFault is truthful.
tonSpaOverTemp(IN := stProcess.rTc1Spa > GVL_SysParameters.rMaxTemp, PT := tGeneral_10s);
IF tonSpaOverTemp.Q THEN
    stFaults.bSpaOverTemp := TRUE;
    _Report(E_FaultId.SpaOverTemp);
END_IF

tonFmOverTemp(IN := stProcess.rTc2FlowMeter > GVL_SysParameters.rMaxTemp,
              PT := tGeneral_10s);
IF tonFmOverTemp.Q THEN
    stFaults.bFlowMeterOverTemp := TRUE;
    _Report(E_FaultId.FlowMeterOverTemp);
END_IF

// External channel is skipped entirely when the external heater is disabled,
// because an unheated line legitimately sits at ambient.
tonExtOverTemp(IN := (stProcess.rTc3External > GVL_SysParameters.rMaxTemp) AND NOT bExternalHeaterOff,
               PT := tGeneral_10s);
IF tonExtOverTemp.Q THEN
    stFaults.bExtOverTemp := TRUE;
    _Report(E_FaultId.ExternalOverTemp);
END_IF

tonDsOverTemp(IN := stProcess.rTc4Delivery > GVL_SysParameters.rMaxTemp,
              PT := tGeneral_10s);
IF tonDsOverTemp.Q THEN
    stFaults.bDownstreamOverTemp := TRUE;
    _Report(E_FaultId.DownstreamOverTemp);
END_IF

//--- HMI communication loss. New in this system; no legacy equivalent. ------
// DISABLED FOR 8.29.26 COMISSIONING
IF NOT bHmiHeartbeatOk THEN
    stFaults.bHmiCommLoss := TRUE;
    _Report(E_FaultId.HmiCommLoss);
END_IF

//=============================================================================
// WARM-UP FAULTS - only while the heater loops are enabled
//=============================================================================
tonWarmup(IN := bTempControlActive, PT := tWarmup);

IF tonWarmup.Q THEN
    IF stProcess.rTc1Spa < GVL_SysParameters.rWarmupTemp THEN
        stFaults.bSpaWarmupTimeout := TRUE;
        _Report(E_FaultId.SpaWarmupTimeout);
    END_IF
    IF stProcess.rTc2FlowMeter < GVL_SysParameters.rWarmupTemp THEN
        stFaults.bFlowmeterWarmupTimeout := TRUE;
        _Report(E_FaultId.FlowMeterWarmupTimeout);
    END_IF
    IF (stProcess.rTc3External < GVL_SysParameters.rWarmupTemp)
       AND NOT bExternalHeaterOff THEN
        stFaults.bExtWarmupTimeout := TRUE;
        _Report(E_FaultId.ExternalWarmupTimeout);
    END_IF
    IF stProcess.rTc4Delivery < GVL_SysParameters.rWarmupTemp THEN
        stFaults.bDownstreamWarmupTimeout := TRUE;
        _Report(E_FaultId.DownstreamWarmupTimeout);
    END_IF
END_IF

//=============================================================================
// EXTERNAL LINE TEMPERATURE - two dedicated checks
//=============================================================================
rtColdStart(CLK := bColdStart);
IF rtColdStart.Q AND NOT bExternalHeaterOff THEN
    rExtTempAtStart := stProcess.rTc3External;
    bExtRiseArmed   := TRUE;
    bExtRiseTested  := FALSE;
END_IF

tonExtWarmupWindow(IN := bExtRiseArmed, PT := tExtRiseTimeout);   // 120 s

IF tonExtWarmupWindow.Q AND NOT bExtRiseTested THEN
    bExtRiseTested := TRUE;
    bExtRiseArmed  := FALSE;
    IF (stProcess.rTc3External - rExtTempAtStart) < GVL_SysParameters.rExtTempMinRise THEN
        stFaults.bExtTempDecoupled := TRUE;
        _Report(E_FaultId.ExternalNoTempRise);
    END_IF
END_IF

tonExtLowAtReady(IN := bReadyReached AND NOT bExternalHeaterOff 
				 AND (stProcess.rTc3External < GVL_SysParameters.rExtMinReadyTemp),
                 PT := tGeneral_10s);      // 10.0 s
IF tonExtLowAtReady.Q THEN
    stFaults.bExtTempLow := TRUE;
    _Report(E_FaultId.ExternalLowAtReady);
END_IF

//=============================================================================
// 4. WATER FAULTS - scoped to the water control sequence
//=============================================================================
// Empty-vessel check. The filter is deliberately much longer during purge,
// because purge repeatedly drains the vessel on purpose and the level would
// otherwise trip this constantly.
tonWaterEmpty(IN := bWaterEmptyFiltered, PT := SEL(bPurgeActive, T#2S, T#30S));

IF tonWaterEmpty.Q THEN
	stFaults.bWaterEmpty := TRUE;
	_Report(E_FaultId.WaterEmpty);
END_IF

// over-filled vessel check
tonWaterOverfill(IN := GVL_IO.biLS2_WaterHighLevel, PT := tFullDelay);

IF tonWaterOverfill.Q THEN
	stFaults.bWaterOverFill := TRUE;
	_Report(E_FaultId.WaterOverFill);
END_IF

// Fill timeout: inlet has been open for the full fill window and the centre
// switch still reports no water. Either the supply is dry or the inlet valve
// is not passing.
tonWaterFill(IN := bWaterFillActive AND NOT bWaterCenterFiltered,
             PT := tWater_15m);
IF tonWaterFill.Q THEN
    stFaults.bWaterFillTimeout := TRUE;
    _Report(E_FaultId.WaterFill);
END_IF

// Regulation fault: the level loop has been asking for water continuously for
// the whole check period. Distinct from the fill timeout - here the level does
// respond, but never satisfies the loop, which points at a leak or a drain
// valve that is not sealing.
(* tonWaterReg(IN := bWaterFillRequest,
            PT := tWater_15m);
IF tonWaterReg.Q THEN
    stFaults.bWaterRegulationFault := TRUE;
    _Report(E_FaultId.WaterRegulation);
END_IF *)

//=============================================================================
// 5. PURGE WATCHDOG - retry once, then fault
//=============================================================================
tonPurge(IN := bPurgeActive, PT := GVL_SysParameters.tPurgeTimeout);

IF tonPurge.Q THEN
	stFaults.bPurgeTimeout := TRUE;
	_Report(E_FaultId.VesselPurgeTimeout);
END_IF

//=============================================================================
// 6. DIFFERENTIAL PRESSURE FAULTS
//=============================================================================
// Downstream too high on entry. Immediate, no filter: this is a go/no-go
// precondition, not a transient.
IF bDiffPressActive AND (stProcess.rPt2Downstream > GVL_SysParameters.rDsHighStartPressure) THEN
    stFaults.bDownstreamStartOverPress := TRUE;
    _Report(E_FaultId.DownstreamStartHigh);
END_IF

// Timeout establishing differential pressure. Same retry-once shape as purge.
tonDiffPress(IN := bDiffPressActive AND NOT bDiffPressReached,
             PT := tDiffPressTimeout);

IF tonDiffPress.Q THEN
	stFaults.bStartDpTimeout := TRUE;
	_Report(E_FaultId.StartupDiffPressTimeout);
END_IF

// Transducer cross-check. Run only when the system is cold and both sides have
// equalised to atmosphere - at that point both transducers must agree, and
// must agree with atmospheric pressure. Any disagreement means one of them has
// drifted, and every downstream flow calculation would inherit the error.
IF eState = E_SystemState.FillWater THEN
    IF (stProcess.rPt2Downstream > GVL_SysParameters.rP3AbsMax)
       OR (stProcess.rPt2Downstream < GVL_SysParameters.rP3AbsMin)
	   OR (ABS(stProcess.rDiffPressureOffset) > GVL_SysParameters.rPtMaxVariance) THEN
        stFaults.bStartDpHardwareFault := TRUE;
        _Report(E_FaultId.StartupDiffPressXCheck);
    END_IF
END_IF

//=============================================================================
// 7. FLOW RATE ERROR
//=============================================================================
// The flow-to-differential-pressure ratio exceeding its calibration maximum
// means the two independent flow measurements disagree - the orifice and the
// SPA pressure drop no longer tell the same story. A differential pressure of
// exactly zero is caught separately because it makes the ratio undefined
// rather than merely large.
// Only meaningful in production above 20% of rated flow; below that the
// differential pressure signal is too small to draw conclusions from.
tonFlowRatio(IN := bSteamFlowing
 			 AND (stProcess.rFlowSetpoint > (0.20 * stProcess.rFlowRated))
			 AND ( (stProcess.rDiffPressure <= 0.0)
			 OR (stProcess.rFlowRatio > GVL_SysParameters.rMaxFlowDpRatio) ),
             PT := tFlowRatioFilter);       // 60 s
IF tonFlowRatio.Q THEN
    stFaults.bFlowFault := TRUE;
    _Report(E_FaultId.FlowRateError);
END_IF

//=============================================================================
// 8. AGGREGATE
//=============================================================================
stFaults.bAnyFault :=
      stFaults.bPowerFault           	 	OR stFaults.bCabinetFlood
   	OR stFaults.bPneumaticLow         	 	OR stFaults.bUpstreamOverPress
   	OR stFaults.bDownstreamOverPress  	 	OR stFaults.bPt1HardwareFault
   	OR stFaults.bPt2HardwareFault     	 	OR stFaults.bSpaOverTemp
   	OR stFaults.bFlowMeterOverTemp    	 	OR stFaults.bExtOverTemp
   	OR stFaults.bDownstreamOverTemp    		OR stFaults.bSpaWarmupTimeout
   	OR stFaults.bFlowmeterWarmupTimeout     OR stFaults.bExtWarmupTimeout
   	OR stFaults.bDownstreamWarmupTimeout    OR stFaults.bExtTempDecoupled
   	OR stFaults.bExtTempLow		    		OR stFaults.bWaterEmpty
   	OR stFaults.bWaterOverFill				OR stFaults.bWaterFillTimeout       		
   	OR stFaults.bWaterRegulationFault		OR stFaults.bPurgeTimeout           		
	OR stFaults.bDownstreamStartOverPress	OR stFaults.bStartDpTimeout     			
	OR stFaults.bFlowFault					OR stFaults.bStartDpHardwareFault		
	OR stFaults.bHmiCommLoss;

bAnyLatchingFault := stFaults.bAnyFault;
bAnyFaultPrev     := stFaults.bAnyFault;

// Capture first-out. Only the first fault in a healthy-to-faulted transition
// is recorded; later faults latch their own bits but do not overwrite the
// reported cause. This is the fix for the legacy behaviour, where the message
// register was overwritten by whichever fault happened to evaluate last in
// the scan, so the operator was routinely shown a downstream consequence
// instead of the actual trigger.
METHOD PRIVATE _Report
VAR_INPUT
    eErrorID		: E_FaultId;
	
END_VAR

VAR
	i				: DINT;
	sErrorString	: STRING(30);
	fbGetSystemTime	: GETSYSTEMTIME;
	fileTime		: T_FILETIME;
END_VAR
IF aActiveFaults[1, UPPER_BOUND(aActiveFaults, 2)] = '' THEN
	sErrorString := TO_STRING(eErrorID);
	FOR i:=LOWER_BOUND(aActiveFaults, 2) TO UPPER_BOUND(aActiveFaults, 2) DO
		IF aActiveFaults[1,i] = sErrorString THEN
			EXIT;
		ELSIF aActiveFaults[1,i] = '' THEN
			// store error
			aActiveFaults[1,i] := sErrorString;
			// grab and store timestamp
			fbGetSystemTime(timeLoDW=>fileTime.dwLowDateTime, timeHiDW=>fileTime.dwHighDateTime );
			aActiveFaults[2,i] := SYSTEMTIME_TO_STRING( FILETIME_TO_SYSTEMTIME( fileTime ) );
			EXIT;
		END_IF
	END_FOR
END_IF
END_METHOD

// Suppress the transducer health checks. The state machine asserts this on
// entry to Fault and drops it once a reset succeeds.
//
// Without it, a genuinely dead transducer re-latches its fault within 250 ms
// of every reset attempt and the operator can never clear the alarm to get to
// maintenance mode. The legacy solved this the same way, by gating those two
// timers on not-being-in-the-fault-stage.
METHOD InhibitSensorHwEval : BOOL
VAR_INPUT
    bInhibit : BOOL;
END_VAR
bSensorHwInhibit := bInhibit;
IF bInhibit THEN
    tonPt1Bad(IN := FALSE);
    tonPt2Bad(IN := FALSE);
END_IF
InhibitSensorHwEval := TRUE;
END_METHOD

// Operator reset. Clears every latch and every filter timer unconditionally,
// then lets the next cycle re-evaluate from scratch. Anything still genuinely
// wrong re-latches immediately and the state machine refuses to leave Fault.
//
// This clears ALL faults, deliberately. The legacy reset cleared only fifteen
// of its bits and left the rest - notably both transducer hardware faults -
// latched until a power cycle. That is not preserved: a fault the operator
// cannot clear and cannot see the reason for is worse than one that re-trips
// honestly on the next scan.
METHOD ResetAll : BOOL
VAR
	i	: DINT;
END_VAR
stFaults.bAnyFault					:= FALSE;
stFaults.bPowerFault          		:= FALSE;
stFaults.bCabinetFlood        		:= FALSE;
stFaults.bPneumaticLow        		:= FALSE;
stFaults.bUpstreamOverPress   		:= FALSE;
stFaults.bDownstreamOverPress 		:= FALSE;
stFaults.bPt1HardwareFault      	:= FALSE;
stFaults.bPt2HardwareFault      	:= FALSE;
stFaults.bSpaOverTemp				:= FALSE;
stFaults.bFlowmeterOverTemp			:= FALSE;
stFaults.bExtOverTemp				:= FALSE;
stFaults.bDownstreamOverTemp		:= FALSE;
stFaults.bSpaWarmupTimeout			:= FALSE;
stFaults.bFlowmeterWarmupTimeout	:= FALSE;
stFaults.bExtWarmupTimeout			:= FALSE;
stFaults.bDownstreamWarmupTimeout	:= FALSE;
stFaults.bExtTempDecoupled			:= FALSE;
stFaults.bExtTempLow				:= FALSE;
stFaults.bWaterEmpty          		:= FALSE;
stFaults.bWaterOverFill				:= FALSE;
stFaults.bWaterFillTimeout          := FALSE;
stFaults.bWaterDrainTimeout         := FALSE;
stFaults.bWaterRegulationFault		:= FALSE;
stFaults.bPurgeTimeout				:= FALSE;
stFaults.bDownstreamStartOverPress	:= FALSE;
stFaults.bStartDpTimeout			:= FALSE;
stFaults.bStartDpHardwareFault		:= FALSE;
stFaults.bFlowFault					:= FALSE;
stFaults.bHmiCommLoss				:= FALSE;

// Filter timers must be cleared too, or a timer already at its preset will
// re-trip on the very next scan regardless of the current input state.
tonPneumaticLow(IN := FALSE);
tonUpstreamHigh(IN := FALSE);
tonDownstreamHigh(IN := FALSE);
tonPt1Bad(IN := FALSE);
tonPt2Bad(IN := FALSE);
tonSpaOverTemp(IN := FALSE);
tonFmOverTemp(IN := FALSE);
tonExtOverTemp(IN := FALSE);
tonDsOverTemp(IN := FALSE);
tonWarmup(IN := FALSE);
tonPurge(IN := FALSE);
tonDiffPress(IN := FALSE);
tonWaterFill(IN := FALSE);
tonWaterReg(IN := FALSE);
tonWaterEmpty(IN := FALSE);
tonExtWarmupWindow(IN := FALSE);
tonExtLowAtReady(IN := FALSE);
tonFlowRatio(IN := FALSE);

bExtRiseArmed       := FALSE;
bExtRiseTested      := FALSE;

FOR i:=LOWER_BOUND(aActiveFaults, 2) TO UPPER_BOUND(aActiveFaults, 2) DO
	aActiveFaults[1,i] := '';
	aActiveFaults[2,i] := '';
END_FOR

InhibitSensorHwEval(FALSE);

ResetAll  := TRUE;
END_METHOD

END_FUNCTION_BLOCK

// ---- POUs/FB_Hmi.TcPOU
FUNCTION_BLOCK FB_Hmi
VAR_INPUT
	eState          		: E_SystemState;
    stProcess       		: ST_ProcessValues;
    stFaults        		: ST_Faults;              // from FB_FaultMonitor
    bReady          		: BOOL;                   // temps in band, ok to flow
	aActiveFaults		: ARRAY[1..2, 1..5] OF STRING(30);
	
    // arPidOutput     : ARRAY[1..6] OF REAL;    // loop outputs 0..100 %
    // arValveActual   : ARRAY[1..4] OF BOOL;    // real valve output states
    // stLimits        : ST_SetpointLimits;      // clamp ranges (defaults ok)
	
END_VAR
VAR_OUTPUT
	// one-cycle command pulses for MAIN / state machine
    bCmdSesOn       	: BOOL;
    bCmdSesOff      	: BOOL;
	bCmdDeliveryOn		: BOOL;
	bCmdDeliveryOff		: BOOL;
    bCmdFaultReset  	: BOOL;
    bCmdFaultAck    	: BOOL;
    bCmdEnterMaint  	: BOOL;
    bCmdExitMaint   	: BOOL;
	bCmdExtHeaterOn		: BOOL;
	bCmdExtHeaterOff	: BOOL;
	bCmdAutofillOn		: BOOL;
	bCmdAutofillOff		: BOOL;
	bCmdDpLoopOn		: BOOL;
	bCmdDpLoopOff		: BOOL;
	bCmdTempLoopOn		: BOOL;
	bCmdTempLoopOff		: BOOL;
	bCmdApplySetpoints	: BOOL;
	
	// heartbeat supervision	
	bHmiCommLoss    : BOOL;  // feed into ST_Faults.bHmiCommLoss
END_VAR

VAR
	// heartbeat supervision
    nLastHeartbeat  : UDINT;
    tonHbTimeout    : TON;
    bFirstCycle     : BOOL := TRUE;
	
	// uptime
    tonUptime       : TON;
    nUptimeSeconds  : UDINT;
    fbTick          : TON;
END_VAR


//=========================== 1. Heartbeat supervision =========================
// Pi increments stCommand.nHmiHeartbeat every poll. If it stops changing
// for T_HMI_HEARTBEAT_TIMEOUT, declare comm loss.
IF (GVL_HMI.stHmiCommand.nHmiHeartbeat = nLastHeartbeat) AND NOT bFirstCycle THEN
	tonHbTimeout(IN := TRUE, PT := GVL_HMI.T_HMI_HEARTBEAT_TIMEOUT);
ELSE
	tonHbTimeout(IN := FALSE);
END_IF

// DISABLED FOR 8.29.26 COMISSIONING
bHmiCommLoss := tonHbTimeout.Q;
nLastHeartbeat := GVL_HMI.stHmiCommand.nHmiHeartbeat;
bFirstCycle := FALSE;

//=========================== 2. Consume command pulses ========================
// Latch each request to the output for exactly one cycle, then clear the
// GVL bit so the Pi never has to write FALSE and a stuck TRUE cannot
// repeat-fire.

// set any new commands
bCmdSesOn  			:= GVL_HMI.stHmiCommand.bSesOn; 
bCmdSesOff     		:= GVL_HMI.stHmiCommand.bSesOff;
bCmdDeliveryOn		:= GVL_HMI.stHmiCommand.bSteamDeliveryOn;
bCmdDeliveryOff		:= GVL_HMI.stHmiCommand.bSteamDeliveryOff;
bCmdFaultReset 		:= GVL_HMI.stHmiCommand.bFaultReset;
bCmdFaultAck   		:= GVL_HMI.stHmiCommand.bFaultAck;
bCmdEnterMaint 		:= GVL_HMI.stHmiCommand.bEnterMaint;
bCmdExitMaint  		:= GVL_HMI.stHmiCommand.bExitMaint;
bCmdExtHeaterOn     := GVL_HMI.stHmiCommand.bExtHeaterOn;
bCmdExtHeaterOff    := GVL_HMI.stHmiCommand.bExtHeaterOff;
bCmdAutofillOn  	:= GVL_HMI.stHmiCommand.bAutofillOn;
bCmdAutofillOff  	:= GVL_HMI.stHmiCommand.bAutofillOff;
bCmdDpLoopOn   		:= GVL_HMI.stHmiCommand.bDpControlOn;
bCmdDpLoopOff   	:= GVL_HMI.stHmiCommand.bDpControlOff;
bCmdTempLoopOn 		:= GVL_HMI.stHmiCommand.bTempControlOn;
bCmdTempLoopOff		:= GVL_HMI.stHmiCommand.bTempControlOff;
bCmdApplySetpoints	:= GVL_HMI.stHmiCommand.bApplySetpoints;

// clear stale cmds
GVL_HMI.stHmiCommand.bSesOn      		:= FALSE;
GVL_HMI.stHmiCommand.bSesOff     		:= FALSE;
GVL_HMI.stHmiCommand.bSteamDeliveryOn 	:= FALSE;
GVL_HMI.stHmiCommand.bSteamDeliveryOff 	:= FALSE;
GVL_HMI.stHmiCommand.bFaultReset 		:= FALSE;
GVL_HMI.stHmiCommand.bFaultAck   		:= FALSE;
GVL_HMI.stHmiCommand.bEnterMaint 		:= FALSE;
GVL_HMI.stHmiCommand.bExitMaint  		:= FALSE;
GVL_HMI.stHmiCommand.bExtHeaterOn   	:= FALSE;
GVL_HMI.stHmiCommand.bExtHeaterOff   	:= FALSE;
GVL_HMI.stHmiCommand.bAutofillOn 		:= FALSE;
GVL_HMI.stHmiCommand.bAutofillOff 		:= FALSE;
GVL_HMI.stHmiCommand.bDpControlOn   	:= FALSE;
GVL_HMI.stHmiCommand.bDpControlOff   	:= FALSE;
GVL_HMI.stHmiCommand.bTempControlOff 	:= FALSE;
GVL_HMI.stHmiCommand.bTempControlOn 	:= FALSE;
GVL_HMI.stHmiCommand.bApplySetpoints	:= FALSE;

// Safety interlock: ignore SES ON during comm-lost or active fault display;
// the state machine makes the final call, this is belt-and-braces.
IF bHmiCommLoss THEN
    bCmdSesOn := FALSE;
END_IF

//=========================== 5. Publish status ================================
GVL_HMI.stHmiStatus.nPlcHeartbeat     := GVL_HMI.stHmiStatus.nPlcHeartbeat + 1;
GVL_HMI.stHmiStatus.nHmiHeartbeatEcho := GVL_HMI.stHmiCommand.nHmiHeartbeat;
GVL_HMI.stHmiStatus.bHmiOnline        := NOT bHmiCommLoss;

GVL_HMI.stHmiStatus.eState       := eState;
GVL_HMI.stHmiStatus.sStateName   := TO_STRING(eState);
GVL_HMI.stHmiStatus.bReady       := bReady;

GVL_HMI.stHmiStatus.stFaults     := stFaults;
GVL_HMI.stHmiStatus.bAlarmActive := stFaults.bAnyFault;
GVL_HMI.stHmiStatus.aActiveFaults := aActiveFaults;
GVL_HMI.stHmiStatus.stProcess    := stProcess;
GVL_HMI.stHmiStatus.sPlcVersion := GVL_HMI.S_PLC_VERSION;

// uptime counter (1 s self-retriggering tick)
fbTick(IN := NOT fbTick.Q, PT := T#1S);
IF fbTick.Q THEN
    nUptimeSeconds := nUptimeSeconds + 1;
END_IF
GVL_HMI.stHmiStatus.nUptimeSeconds := nUptimeSeconds;

END_FUNCTION_BLOCK

// ---- POUs/FB_PressureControl.TcPOU
//=============================================================================
// FB_PressureControl | DRAFT 8.2.26 - NOT YET VERIFIED ON HARDWARE
//-----------------------------------------------------------------------------
// All closed-loop heater control. 
//
// Each loop has two parts:
//   PID  -> a demand in percent
//   PWM  -> that percent turned into on/off time inside a fixed period
//
// LOOP MAP:
//   [1] Boiler / upstream pressure  PT1 -> H1   PID1
//   [2] SPA (purifier) temperature  TC1 -> H2   PID2
//   [3] Flow meter temperature      TC2 -> H3   PID3
//   [4] External line heater        TC3 -> H4   bang-bang + hysteresis, NOT PID.
//
// BOILER PRESSURE SETPOINT (loop 1) has three sources, in priority order:
//   1. PurgeVessel state -> purge target pressure
//   2. SPA not yet flushed -> PT3 + initial dP (100 Torr)
//   3. normal -> PT2 + target dP + tuning offset
// In cases 1 and 2 the PWM period is doubled while the max on-time stays
// fixed, which is how the legacy capped the boiler heater at 50 % duty.
// Once flushed, the setpoint is RAMPED at 1 Torr per 0.5 s instead of stepped.
// Drives NO coil directly. Outputs heater demands; FB_OutputHandler is the
// single writer and still gates everything on state.
//
// DEVIATIONS FROM THE LEGACY (all deliberate, all flagged inline):
//   * gains are re-expressed in engineering units (%/Torr, %/degC) - see
//     GVL_SysParameters for the conversion arithmetic. RETUNE ON THE BENCH.
//   * setpoint ramp clamps at the target instead of dithering +/-1 Torr.
//   * ramp is preloaded from live PT1 on enable (legacy did this only on the
//     hot-restart path, rung 85).
//   * derivative acts on the measurement, not the error, to kill setpoint kick.
//   * SPA heater gets a hard over-temperature cut. The legacy had none.
//   * external heater gets turn-off hysteresis. The legacy had none.
//=============================================================================
FUNCTION_BLOCK FB_PressureControl
VAR_INPUT
    bEnable             : BOOL;              // FB_StateMachine.bControlEnable
    eState              : E_SystemState;     // needed to detect PurgeVessel & SpaFlush
    bDpControlOff       : BOOL;              // HMI/maint: suspend loop 1
    bTempControlOff     : BOOL;              // HMI/maint: suspend loop 2
    bExtHeaterEnable    : BOOL;              // HMI: external heater allowed
    stProcess           : ST_ProcessValues;  // scaled PVs
    stSetpoints         : ST_HmiSetpoints;   // operator setpoints, already clamped by FB_Hmi
    rTargetDiffPressure : REAL;              // [Torr] from FB_FlowCalcs
	bFlushed            : BOOL;
	bSpaPressurized		: BOOL;				 // SPA at pressure
END_VAR
VAR_OUTPUT
    // --- heater demands -> FB_OutputHandler (single writer) ---------------
    qH1_UpstreamHeater  : BOOL;              // H1
    qH2_SpaHeater       : BOOL;              // H2
    qH3_FlowmeterHeater : BOOL;              // H3
    qH4_ExternalHeater  : BOOL;              // H4

    // --- HMI / diagnostics -------------------------------------------------
    arOutputPct         : ARRAY[1..4] OF REAL; // loop demand 0..100 %
    rBoilerSpTarget     : REAL;                // where we want to be
    rBoilerSpActive     : REAL;                // ramped SP fed to PID1
    bDiffPressReached   : BOOL; 
END_VAR
VAR
    // --- edges / gating ----------------------------------------------------
    rtrigEnable         : R_TRIG;
    bPurging            : BOOL;

    // --- PID sample-rate gate (legacy K5 = 0.05 s) -----------------
    fbSampleTick        : TON;
    bSample             : BOOL;
    rDt                 : REAL;              // [s] sample interval as a real

    // --- loop 1 setpoint generation ----------------------------------------
    fbRampTick          : TON;
    tPwmPeriod1         : TIME;
    rDutyCap1           : REAL;

    // --- per-loop PID state (index = legacy PID number) --------------------
    arIntegral          : ARRAY[1..4] OF REAL;
    arPrevPv            : ARRAY[1..4] OF REAL;
    arPrimed            : ARRAY[1..4] OF BOOL;

    // --- per-loop PWM state -------------------------------------------------
    arPwmTimer          : ARRAY[1..4] OF TON;
    arPwmDutyLatched    : ARRAY[1..4] OF REAL;

    i                   : INT;
END_VAR

//============================================================================
// 0. SAFE STATE WHEN DISABLED
//============================================================================
// Everything off, every integrator and timer cleared, so a re-enable always
// starts from a known state instead of resuming with stale wind-up.
rtrigEnable(CLK := bEnable);

IF NOT bEnable THEN
    FOR i := 1 TO 4 DO
        ResetLoop(nLoop := i);
    END_FOR
    qH1_UpstreamHeater  := FALSE;
    qH2_SpaHeater       := FALSE;
    qH3_FlowmeterHeater := FALSE;
    qH4_ExternalHeater  := FALSE;
    bDiffPressReached   := FALSE;
    fbSampleTick(IN := FALSE);
    fbRampTick(IN := FALSE);
    RETURN;
END_IF

// Preload the ramp from wherever the boiler actually is, so the first
// enable does not walk up from zero
IF rtrigEnable.Q THEN
    rBoilerSpActive := stProcess.rPt1Upstream;
END_IF

bPurging := (eState = E_SystemState.PurgeVessel);

//============================================================================
// 1. PID SAMPLE TICK
//============================================================================
// The PID math runs on a fixed interval, not every task cycle, so rDt is a
// known constant. tPidSampleTime MUST be a whole multiple of the task cycle.
fbSampleTick(IN := NOT fbSampleTick.Q, PT := GVL_SysParameters.tPidSampleTime);
bSample := fbSampleTick.Q;
rDt     := UDINT_TO_REAL(TIME_TO_UDINT(GVL_SysParameters.tPidSampleTime)) * 0.001;

//============================================================================
// 2. LOOP 1 SETPOINT SELECTION
//============================================================================
IF bPurging THEN
    // Hold the boiler just above atmosphere so FB_Purge can cycle the drain.
    // Uses the same parameter FB_Purge bands around - keep these two together.
    rBoilerSpTarget := GVL_SysParameters.rPurgeTargetPressure;

ELSIF eState = E_SystemState.InitMain AND NOT bFlushed THEN
    // SPA not flushed yet: PT3 + initial dP. The state machine cycles the
    // boiler across this setpoint N times to flush the SPA before release.
	IF NOT bSpaPressurized THEN
		rBoilerSpTarget := GVL_SysParameters.rAtmosphericPressure + GVL_SysParameters.rIniDeltaPressure;
	ELSE
		rBoilerSpTarget := GVL_SysParameters.rAtmosphericPressure + GVL_SysParameters.rIniDeltaPressure/2;
	END_IF
    

ELSE
    // Normal running: hold PT1 a target differential above PT2.
	rTargetDiffPressure := _TargetDiffPressure(rFlowSp := GVL_HMI.stHmiSetpoints.rSetFlow);
	
    rBoilerSpTarget := stProcess.rPt2Downstream + rTargetDiffPressure + GVL_SysParameters.rPspGainOffset;
END_IF

//============================================================================
// 3. LOOP 1 SETPOINT RAMP
//============================================================================
// Before the flush the setpoint is applied immediately; after it, walk the
// active setpoint toward the target one step at a time so a flow change does
// not slam the boiler.
IF NOT bFlushed THEN
    rBoilerSpActive := rBoilerSpTarget;
    fbRampTick(IN := FALSE);
ELSE
    fbRampTick(IN := NOT fbRampTick.Q, PT := GVL_SysParameters.tSpRampInterval);
    IF fbRampTick.Q THEN
        IF rBoilerSpActive < rBoilerSpTarget THEN
            rBoilerSpActive := MIN(rBoilerSpActive + GVL_SysParameters.rSpRampStep, rBoilerSpTarget);
        ELSIF rBoilerSpActive > rBoilerSpTarget THEN
            rBoilerSpActive := MAX(rBoilerSpActive - GVL_SysParameters.rSpRampStep, rBoilerSpTarget);
        END_IF
    END_IF
END_IF

// "Target reached" - cancels the startup differential-pressure watchdog in
// FB_StateMachine. Compared against the target WITHOUT the tuning offset
bDiffPressReached := (stProcess.rPt1Upstream >= (rBoilerSpTarget - GVL_SysParameters.rPspGainOffset));

//============================================================================
// 4. LOOP 1  -  BOILER PRESSURE -> H1
//============================================================================
// Slow PWM period while purging or before the flush. The max on-time is
// fixed, so doubling the period is what halves the duty ceiling to 50 %.
IF bPurging OR NOT bFlushed THEN
    tPwmPeriod1 := GVL_SysParameters.tPid1PwmPeriodSlow;
	rDutyCap1 := 50.0;
ELSE
    tPwmPeriod1 := GVL_SysParameters.tPid1PwmPeriod;
	rDutyCap1 := 100.0 * UDINT_TO_REAL(TIME_TO_UDINT(GVL_SysParameters.tPid1MaxOnTime))
			   / UDINT_TO_REAL(TIME_TO_UDINT(tPwmPeriod1));
	rDutyCap1 := LIMIT(0.0, rDutyCap1, 80.0);
END_IF



IF bDpControlOff THEN
    ResetLoop(nLoop := 1);
    qH1_UpstreamHeater := FALSE;
ELSE
    IF bSample THEN
        arOutputPct[1] := RunPid(nLoop     := 1,
                                 rSp       := rBoilerSpActive,
                                 rPv       := stProcess.rPt1Upstream,
                                 rKp       := GVL_SysParameters.rPid1_Kp,
                                 rTi       := GVL_SysParameters.rPid1_Ti,
                                 rTd       := GVL_SysParameters.rPid1_Td,
                                 rOutMin   := 0.0,
                                 rOutMax   := rDutyCap1,
                                 rDt       := rDt);
    END_IF
    qH1_UpstreamHeater := RunPwm(nLoop    := 1,
                                 rDutyPct := arOutputPct[1],
                                 tPeriod  := tPwmPeriod1);

    // hard over-temperature cut. FB_FaultMonitor will also trip on this, 
	// but the heater should not wait for the state machine to react.						 
	IF stProcess.rPt1Upstream >= GVL_SysParameters.rUpstreamMaxPressure THEN 
		qH1_UpstreamHeater := FALSE; 
	END_IF
END_IF

//============================================================================
// 5. LOOP 2  -  SPA TEMPERATURE -> H2
//============================================================================
IF bTempControlOff THEN
    ResetLoop(nLoop := 2);
    qH2_SpaHeater := FALSE;
ELSE
    IF bSample THEN
        arOutputPct[2] := RunPid(nLoop     := 2,
                                 rSp       := GVL_SysParameters.rSpaTempSp,
                                 rPv       := stProcess.rTc1Spa,
                                 rKp       := GVL_SysParameters.rPid2_Kp,
                                 rTi       := GVL_SysParameters.rPid2_Ti,
                                 rTd       := GVL_SysParameters.rPid2_Td,
                                 rOutMin   := 0.0,
                                 rOutMax   := 100.0,
                                 rDt       := rDt);
    END_IF
    qH2_SpaHeater := RunPwm(nLoop    := 2,
                            rDutyPct := arOutputPct[2],
                            tPeriod  := GVL_SysParameters.tPid2PwmPeriod);

    // hard over-temperature cut. FB_FaultMonitor will also trip on this, 
	// but the heater should not wait for the state machine to react.
    IF stProcess.rTc1Spa >= GVL_SysParameters.rMaxTemp THEN
        qH2_SpaHeater := FALSE;
    END_IF
END_IF

//============================================================================
// 6. LOOP 3  -  FLOW METER TEMPERATURE -> H3
//============================================================================
IF bSample THEN
    arOutputPct[3] := RunPid(nLoop     := 3,
                             rSp       := GVL_SysParameters.rFlowMeterTempSp,
                             rPv       := stProcess.rTc2FlowMeter,
                             rKp       := GVL_SysParameters.rPid3_Kp,
                             rTi       := GVL_SysParameters.rPid3_Ti,
                             rTd       := GVL_SysParameters.rPid3_Td,
                             rOutMin   := 0.0,
                             rOutMax   := 100.0,
                             rDt       := rDt);
END_IF
qH3_FlowmeterHeater := RunPwm(nLoop    := 3,
                              rDutyPct := arOutputPct[3],
                              tPeriod  := GVL_SysParameters.tPid5PwmPeriod);

// The flow meter heater is inhibited whenever TC4 is at or above the cutout.
IF stProcess.rTc4Delivery >= GVL_SysParameters.rDeliveryTempCutout THEN
    qH3_FlowmeterHeater := FALSE;
END_IF

//============================================================================
// 7. LOOP 4  -  EXTERNAL LINE HEATER -> H4
//============================================================================
IF NOT bExtHeaterEnable THEN
    qH4_ExternalHeater := FALSE;
ELSIF stProcess.rTc3External <= GVL_SysParameters.rExtHeaterTempSp THEN
    qH4_ExternalHeater := TRUE;
ELSIF stProcess.rTc3External > GVL_SysParameters.rExtHeaterTempSp THEN
    qH4_ExternalHeater := FALSE;
END_IF
// else: inside the hysteresis band, hold the last state
arOutputPct[4] := SEL(qH4_ExternalHeater, 0.0, 100.0);

METHOD _TargetDiffPressure : REAL
VAR_INPUT
    rFlowSp     : REAL;   // set flow rate
END_VAR
VAR        
    rQtotal 	: REAL;
	
	// target dp calculation
	rOrificeA1				: REAL := 0.05946087;	// main orifice coefficient
	rOrificeB1				: REAL := 0.0;			// main orifice offset
	rPtMinTorr				: REAL := 50;			// minimum torr to enable calculated flow
END_VAR
rQtotal := rFlowSp + stProcess.rCondensateFlow + rOrificeB1;

IF stProcess.rPt2Downstream > rPtMinTorr THEN
    _TargetDiffPressure := (rQtotal * rQtotal)/(rOrificeA1 * rOrificeA1)/stProcess.rPt2Downstream;
ELSE
    _TargetDiffPressure := 0.0;
END_IF
END_METHOD

//=============================================================================
// ResetLoop
//-----------------------------------------------------------------------------
// Clears every piece of memory belonging to one loop: integral accumulator,
// derivative history, PWM timer and latched duty, published output.
// Called when the loop is disabled so a re-enable never inherits wind-up or
// a stale pulse width.
//=============================================================================
METHOD PRIVATE ResetLoop
VAR_INPUT
    nLoop : INT;
END_VAR
IF (nLoop < 1) OR (nLoop > 4) THEN
    RETURN;
END_IF

arIntegral[nLoop]       := 0.0;
arPrevPv[nLoop]         := 0.0;
arPrimed[nLoop]         := FALSE;
arPwmDutyLatched[nLoop] := 0.0;
arPwmTimer[nLoop](IN := FALSE);
arOutputPct[nLoop]      := 0.0;
END_METHOD

//=============================================================================
// RunPid
//-----------------------------------------------------------------------------
// Standard (ISA) positional PID, output in percent.
//
//   out = Kp * e  +  (Kp/Ti) * INTEGRAL(e)  -  Kp * Td * d(PV)/dt
//
// Derivative acts on the MEASUREMENT, not the error, so a setpoint change
// does not produce a derivative spike.
//
// Anti-windup: the integral accumulator is clamped to the output range. This
// is the same trick as legacy rung 456 ("freeze integral if over"), which
// clamped the PID bias word to the output maximum.
//
// State lives in the FB's arrays, indexed by nLoop, so one method serves
// every loop. Call at the sample rate only - it uses rDt, not the task cycle.
//=============================================================================
METHOD PRIVATE RunPid : REAL
VAR_INPUT
    nLoop   : INT;      // 1..4, index into the state arrays
    rSp     : REAL;     // setpoint, engineering units
    rPv     : REAL;     // process value, same units
    rKp     : REAL;     // proportional gain [% per engineering unit]
    rTi     : REAL;     // integral / reset time [s]. 0 disables integral action
    rTd     : REAL;     // derivative / rate time [s]. 0 disables derivative
    rOutMin : REAL;     // output floor [%]
    rOutMax : REAL;     // output ceiling [%]
    rDt     : REAL;     // sample interval [s]
END_VAR
VAR
    rError  : REAL;
    rProp   : REAL;
    rDeriv  : REAL;
    rOut    : REAL;
END_VAR
IF (nLoop < 1) OR (nLoop > 4) OR (rDt <= 0.0) THEN
    RunPid := 0.0;
    RETURN;
END_IF

rError := rSp - rPv;

//--- proportional ------------------------------------------------------------
rProp := rKp * rError;

//--- integral ----------------------------------------------------------------
IF rTi > 0.0 THEN
    arIntegral[nLoop] := arIntegral[nLoop] + (rKp / rTi) * rError * rDt;
    // clamp to the output range: prevents wind-up while saturated
    arIntegral[nLoop] := LIMIT(rOutMin, arIntegral[nLoop], rOutMax);
ELSE
    arIntegral[nLoop] := 0.0;
END_IF

//--- derivative on measurement ------------------------------------------------
// Skipped on the first sample after a reset, when arPrevPv is meaningless.
IF (rTd > 0.0) AND arPrimed[nLoop] THEN
    rDeriv := -rKp * rTd * (rPv - arPrevPv[nLoop]) / rDt;
ELSE
    rDeriv := 0.0;
END_IF
arPrevPv[nLoop] := rPv;
arPrimed[nLoop] := TRUE;

//--- sum and clamp ------------------------------------------------------------
rOut   := rProp + arIntegral[nLoop] + rDeriv;
RunPid := LIMIT(rOutMin, rOut, rOutMax);
END_METHOD

//=============================================================================
// RunPwm
//-----------------------------------------------------------------------------
// Time-proportioned output: turns a 0..100 % demand into a digital heater
// command with a fixed period. 
//
// The demand is LATCHED at each period boundary. Without this the
// on-time would move underneath an in-progress pulse.
//
// Must be called EVERY task cycle - the period timer only advances when it
// is called. Resolution is one task cycle (10 ms), so a 2 s period gives
// 0.5 % granularity.
//=============================================================================
METHOD PRIVATE RunPwm : BOOL
VAR_INPUT
    nLoop    : INT;     // 1..4, index into the timer array
    rDutyPct : REAL;    // demand 0..100 %
    tPeriod  : TIME;    // PWM period
END_VAR
VAR
    nPeriodMs : UDINT;
    nOnMs     : UDINT;
    rDuty     : REAL;
END_VAR
nPeriodMs := TIME_TO_UDINT(tPeriod);

IF (nLoop < 1) OR (nLoop > 4) OR (nPeriodMs = 0) THEN
    RunPwm := FALSE;
    RETURN;
END_IF

//--- free-running period timer -----------------------------------------------
// IN := NOT Q self-restarts the TON: Q is true for one cycle, which drops IN,
// which clears ET. Costs one task cycle per period (0.5 % at 2 s).
arPwmTimer[nLoop](IN := NOT arPwmTimer[nLoop].Q, PT := tPeriod);

//--- latch the demand once per period ----------------------------------------
// ET is only zero at a period boundary (and on the very first call), so this
// refreshes the on-time exactly once per pulse and never mid-pulse.
IF arPwmTimer[nLoop].ET = T#0S THEN
    arPwmDutyLatched[nLoop] := rDutyPct;
END_IF

rDuty := LIMIT(0.0, arPwmDutyLatched[nLoop], 100.0);

//--- resolve the pulse --------------------------------------------------------
IF rDuty <= 0.0 THEN
    RunPwm := FALSE;
ELSIF rDuty >= 100.0 THEN
    // Special-cased so a saturated loop holds the coil solid instead of
    // dropping out for the single cycle it takes the timer to roll over.
    RunPwm := TRUE;
ELSE
    nOnMs  := REAL_TO_UDINT(rDuty * 0.01 * UDINT_TO_REAL(nPeriodMs));
    RunPwm := TIME_TO_UDINT(arPwmTimer[nLoop].ET) < nOnMs;
END_IF
END_METHOD

END_FUNCTION_BLOCK

// ---- POUs/FB_Purge.TcPOU
//=============================================================================
// FB_Purge | VERIFIED 8.2.26 DA
//-----------------------------------------------------------------------------
//
// MECHANISM - it is a repeating DRAIN / EQUILIBRATE cycle, not a one-shot:
//   * A pressure band is built around the target setpoint:
//       upper = TSP + band 
//       lower = TSP - band 
//   * Purge only proceeds while upstream pressure is inside that band.
//   * Cycle, gated by "OK to purge" latch:
//       1. Open drain valve SV1 for tDrainOpen 
//       2. Close SV1, wait tEquilibrate to let water settle and for the boiler
//			pressuer loop to raise the upstream pressure to within the range
//       3. If the EMPTY switch (LS3) now reads empty -> purge complete.
//          Otherwise, if still in band, re-open SV1 and repeat.
//   * Overall watchdog: if the cycle runs longer than tPurgeTimeout -> bPurgeFault
//   * After complete: water fill is allowed and the state machine advances
//     to SetDiffPressure
//
// Reports intent only:
//   qDrainValve -> FB_OutputHandler -> GVL_IO.qxSv1Drain (single writer).
//   bPurgeComplete -> FB_StateMachine (S11 -> S13 transition).
//   bPurgeTimeout  -> FB_FaultMonitor (latches the fault, like every other).
//=============================================================================
FUNCTION_BLOCK FB_Purge
VAR_INPUT
    bEnable         		: BOOL;    // TRUE while state = PurgeVessel
    rUpstreamPress  		: REAL;    // upstream pressure [Torr]
    bEmptyFiltered  		: BOOL;    // filtered LS3 empty switch
END_VAR             		
VAR_OUTPUT          		
    qDrainValve     		: BOOL;    // -> FB_OutputHandler -> SV1 drain
    bPurgeComplete  		: BOOL;    // -> state machine
    bPurgeTimeout   		: BOOL;    // -> FaultMonitor Momentary report
    bInPressureBand 		: BOOL;    // diagnostic: pressure within purge band
END_VAR
VAR
    bOkToPurge      		: BOOL;    // "OK to purge" drain-phase latch
    bTimeoutRetryUsed		: BOOL;	   //
	rPressureBandUpper      : REAL;    // 
    rPressureBandLower      : REAL;    // 

    tonDrainOpen    		: TON;     // valve-open dwell
    tonEquilibrate  		: TON;     // valve-closed settle
    tonPurgeTimeout 		: TON;     // overall watchdog
END_VAR

IF NOT bEnable THEN
    qDrainValve       := FALSE;
    bOkToPurge        := FALSE;
    bPurgeComplete    := FALSE;
    bPurgeTimeout     := FALSE;
    bTimeoutRetryUsed := FALSE;
    tonDrainOpen(IN := FALSE);
    tonEquilibrate(IN := FALSE);
    tonPurgeTimeout(IN := FALSE);
    RETURN;
END_IF
// NOTE: the state machine must hold bEnable TRUE for the WHOLE PurgeVessel
// state. Dropping it the moment purge finishes lands here and wipes
// bPurgeComplete, which would restart the blowdown.

//--- pressure band (rung 102) ------------------------------------------------
// Parameters are owned by whoever computes the atmospheric reference. This FB
// only reads them.
rPressureBandUpper := GVL_SysParameters.rPurgeTargetPressure + GVL_SysParameters.rPurgeBand;
rPressureBandLower := GVL_SysParameters.rPurgeTargetPressure - GVL_SysParameters.rPurgeBand;
bInPressureBand    := (rUpstreamPress >= rPressureBandLower)
                  AND (rUpstreamPress <  rPressureBandUpper);

//--- latch the cycle once the boiler reaches the band (rung 105) -------------
// Latch only. The valve stays shut; the first thing that happens is a settle.
IF (NOT bOkToPurge) AND (NOT bPurgeComplete) AND bInPressureBand THEN
    bOkToPurge := TRUE;
END_IF

IF bOkToPurge THEN
    //--- drain-open dwell (rungs 106-107) ------------------------------------
    tonDrainOpen(IN := qDrainValve, PT := GVL_SysParameters.tDrainOpen);
    IF tonDrainOpen.Q THEN
        qDrainValve := FALSE;
    END_IF

    //--- settle dwell, runs whenever the valve is shut (rung 108) ------------
    // Self-rearming: opening the valve drops IN, which resets it.
    tonEquilibrate(IN := NOT qDrainValve, PT := GVL_SysParameters.tEquilibrate);

    //--- end of each settle: done, or blow down again (rungs 109-110) --------
    IF tonEquilibrate.Q THEN
        IF bEmptyFiltered THEN
            bOkToPurge     := FALSE;
            bPurgeComplete := TRUE;
            qDrainValve    := FALSE;
        ELSIF bInPressureBand THEN
            qDrainValve := TRUE;
        END_IF
        // else: pressure fell out of band - hold here until the boiler
        // loop brings it back, then open. (Legacy rung 110 does the same.)
    END_IF

    //--- watchdog, one free retry (rungs 111-113) ----------------------------
    tonPurgeTimeout(IN := TRUE, PT := GVL_SysParameters.tPurgeTimeout);
    IF tonPurgeTimeout.Q THEN
        IF bTimeoutRetryUsed THEN
            bPurgeTimeout := TRUE;
        ELSE
            bTimeoutRetryUsed := TRUE;
            tonPurgeTimeout(IN := FALSE);   // restart for the second window
        END_IF
    END_IF
ELSE
    qDrainValve := FALSE;                   // rung 104
    tonDrainOpen(IN := FALSE);
    tonEquilibrate(IN := FALSE);
    tonPurgeTimeout(IN := FALSE);
    bPurgeTimeout := FALSE;
END_IF

END_FUNCTION_BLOCK

// ---- POUs/FB_SpaFlush.TcPOU
FUNCTION_BLOCK FB_SpaFlush // VERIFIED 8.9.26 DASH
VAR_INPUT
    bEnable         : BOOL;   // TRUE while in SteamPrecheck
    bReset          : BOOL;   // clear counter + completion
    rUpstreamPress  : REAL;   // PT1 [Torr]
    rAtmPressure	: REAL;   // crossing threshold [Torr] 
END_VAR

VAR_OUTPUT
    bSpaFlushed     : BOOL;   // -> pressure loop mode + state machine (legacy C10)
    nCrossings      : UINT;   // -> HMI progress display   (legacy V2557)
    bSpaPressurized : BOOL;   // diagnostic: above threshold, awaiting the fall
END_VAR

VAR
    tonConfirm      	: TON;    // falling-edge confirm dwell (legacy T6)
	tConfirmDelay		: TIME := T#10S;
    rSpaFlushPressure	: REAL;
	nFlushCycles		: UINT := 20;
END_VAR

// reset
IF bReset THEN
    nCrossings  := 0;
    bSpaPressurized := FALSE;
    bSpaFlushed := FALSE;
    tonConfirm(IN := FALSE);
    RETURN;
END_IF

IF (NOT bEnable) OR bSpaFlushed THEN
	// idle
	bSpaPressurized := FALSE;
    tonConfirm(IN := FALSE);
    RETURN;
END_IF

IF bEnable THEN
	// set pressure target
	rSpaFlushPressure := rAtmPressure + GVL_SysParameters.rIniDeltaPressure;

	// latch when pressure above target
	IF rUpstreamPress >= rSpaFlushPressure THEN
		bSpaPressurized := TRUE;
	END_IF

	// confirm fall when pressure drops below setpoint for time delay
	tonConfirm(IN := bSpaPressurized AND (rUpstreamPress < rSpaFlushPressure),
			   PT := tConfirmDelay);

	// increment count on timer completion
	IF tonConfirm.Q THEN
		nCrossings := nCrossings + 1;
		bSpaPressurized := FALSE;
		tonConfirm(IN := FALSE);
	END_IF
	
	// successful flush
	IF nCrossings >= nFlushCycles THEN
		bSpaFlushed := TRUE;
		bSpaPressurized := FALSE;
		tonConfirm(IN := FALSE);
	END_IF
END_IF

END_FUNCTION_BLOCK

// ---- POUs/FB_StateMachine.TcPOU
FUNCTION_BLOCK FB_StateMachine
VAR_INPUT
    stFaults    		: ST_Faults;
    stHmiSetpoints 		: ST_HmiSetpoints;
	stProcessValues		: ST_ProcessValues;
	bFillComplete		: BOOL;
	bPurgeComplete		: BOOL;
	bSpaFlushed			: BOOL;
	bDpReached			: BOOL;
END_VAR
VAR_OUTPUT
	// system state
    eState           : E_SystemState := E_SystemState.InitController;
    // enable flags for downstream FBs
	eWaterFillMode 	 : E_WaterFillMode;   	// water fill mode startup/autofill/idle
	bControlEnable   : BOOL;   				// PID pressure/temp loops may run
    bPurgeEnable     : BOOL;   				// vessel purge sequence active
	bSpaFlushEnable	 : BOOL;				// enable SPA flush sequence
	bSpaFlushReset	 : BOOL;				// reset SPA flush fb
	bDeliveryEnable	 : BOOL;				// enable steam delivery
	bAutofillEnable	 : BOOL := TRUE;		// enable water autofill during running states
	bExtHeaterEnable : BOOL;				// enable external heater
	bDpLoopEnable	 : BOOL := TRUE;		// enable dp loop
	bTempLoopEnable	 : BOOL := TRUE;		// enable temp loop
    bReady           : BOOL;   				// green Ready: in SteamFlowing, in-band, no faults
    bInStartup       : BOOL;   				// TRUE for any Init* state
	bColdStart		 : BOOL;				// true if most recent startup was cold
END_VAR
VAR
    // --- request flags set by methods, cleared when serviced ---
    bReqStart        : BOOL;
    bReqStop         : BOOL;
    bReqMaint        : BOOL;
    bReqExitMaint    : BOOL;
    bReqFault        : BOOL;
    bReqFaultReset   : BOOL;
	bReqDelivery	 : BOOL;
    // --- state entry detection (rising edge of a new state) ---
    eStatePrev       : E_SystemState;
    bEntry           : BOOL;   // TRUE on the first cycle of the current state

	// --- tmrs for ready condition ---
	tmrReadyMake	: TON;
	tmrReadyBreak	: TON;
	tMakeOrBreak	: TIME := T#1M;

	
END_VAR

//=========================== entry-edge detection ============================
bEntry := (eState <> eStatePrev);
eStatePrev := eState;

//=========================== reset on entry detection ========================
IF bEntry THEN	
	// do something
END_IF

//=========================== global fault override ===========================
// A latching fault forces Fault from ANY state except when already resetting.
IF bReqFault AND (eState <> E_SystemState.Fault) THEN
    eState := E_SystemState.Fault;
    bEntry := TRUE;
END_IF
bReqFault := FALSE;

//=========================== default enable flags ============================
// Recomputed every cycle; each state turns on what it needs below.
eWaterFillMode 		:= E_WaterFillMode.Idle;
bControlEnable  	:= FALSE;
bPurgeEnable    	:= FALSE;
bSpaFlushEnable 	:= FALSE;
bSpaFlushReset  	:= FALSE;
bDeliveryEnable 	:= FALSE;
bReady          	:= FALSE;
bInStartup      	:= FALSE;

// reset retained vars
IF eState <> E_SystemState.SteamFlowing THEN RequestDelivery(FALSE); END_IF


//================================ STATE MACHINE ==============================
CASE eState OF

    //--------------------------------------------------------------------
    E_SystemState.InitController:   // S0 : one-shot init, then idle
    //--------------------------------------------------------------------
        IF bEntry THEN
            // TODO: seed thresholds from GVL_Params here if they differ per unit
            ;
        END_IF
        eState := E_SystemState.SesOff;

    //--------------------------------------------------------------------
    E_SystemState.SesOff:           // S70 : SES off, idle / standby
    //--------------------------------------------------------------------
        IF bReqMaint THEN
            eState := E_SystemState.Maintenance;
        ELSIF stFaults.bAnyFault THEN
			bReqFault := TRUE;
		ELSIF bReqStart AND NOT stFaults.bHmiCommLoss THEN
            eState := E_SystemState.CheckIfHot;
        END_IF

    //--------------------------------------------------------------------
    E_SystemState.CheckIfHot:       // S10 : hot-restart shortcut vs cold start
    //--------------------------------------------------------------------
        // SPA warm (TC1 within band) AND steam flow already > x%*RatedFlow -> jump to SteamFlowing.
        // Otherwise cold start -> fill water
        bInStartup := TRUE;
        IF _IsSpaWarm() AND (_FlowPercent() > GVL_SysParameters.rHotRestartFlowPct) THEN
            eState := E_SystemState.SteamFlowing;
			bColdStart := FALSE;
		ELSE
            eState := E_SystemState.FillWater;
			bColdStart := TRUE;
			bSpaFlushReset := TRUE;
        END_IF

    //--------------------------------------------------------------------
    E_SystemState.FillWater:    // S20 : fill water
    //--------------------------------------------------------------------
        bInStartup      := TRUE;
        eWaterFillMode 	:= E_WaterFillMode.StartupFill;

        IF bReqStop THEN
            eState := E_SystemState.SesOff;
        ELSIF stFaults.bAnyFault THEN
            bReqFault := TRUE;  
        ELSIF bFillComplete THEN
			IF GVL_HMI.stHmiSetpoints.bSetPurgeOnStartup THEN 
				eState := E_SystemState.PurgeVessel;
			ELSE 
				eState := E_SystemState.SetDiffPressure; 
			END_IF
        END_IF

    //--------------------------------------------------------------------
    E_SystemState.PurgeVessel:  // S30 : purge vessel
    //--------------------------------------------------------------------
        bInStartup   := TRUE;
        bPurgeEnable := TRUE;
		bControlEnable := TRUE;

		// Blowdown first, refill second
		IF bPurgeComplete THEN
			eWaterFillMode := E_WaterFillMode.StartupFill;   // legacy rung 114
		ELSE
			eWaterFillMode := E_WaterFillMode.Idle;          // legacy rung 103: "do not fill water until purge complete"
		END_IF

        IF bReqStop THEN
            eState := E_SystemState.SesOff;
        ELSIF stFaults.bAnyFault THEN
            bReqFault := TRUE;
        ELSIF bPurgeComplete AND bFillComplete THEN
            eState := E_SystemState.SetDiffPressure;
        END_IF

    //--------------------------------------------------------------------
    E_SystemState.SetDiffPressure: // S40 : establish differential pressure
    //--------------------------------------------------------------------
        bInStartup     := TRUE;
        bControlEnable := TRUE;   // dP PID runs to bring differential up

        IF bReqStop THEN
            eState := E_SystemState.SesOff;
		ELSIF stFaults.bAnyFault THEN
            bReqFault := TRUE;    // legacy DS start-high -> S10
        ELSIF bDpReached THEN
            eState := E_SystemState.InitMain;
        END_IF

    //--------------------------------------------------------------------
    E_SystemState.InitMain:         // S50 : final checks before flow
    //--------------------------------------------------------------------
		IF bEntry THEN
			IF GVL_HMI.stHmiSetpoints.rSetFlow = 0 THEN
				GVL_HMI.stHmiSetpoints.rSetFlow := 10;
			END_IF
		END_IF

		bInStartup     := TRUE;
		bControlEnable := TRUE;
		bSpaFlushEnable := TRUE;
		eWaterFillMode := E_WaterFillMode.RunningAutofill;
	
		IF bReqStop THEN
			eState := E_SystemState.SesOff;
		ELSIF stFaults.bAnyFault THEN
			bReqFault := TRUE;
		ELSIF bSpaFlushed AND _TempsInBand() AND _FlowInBand() THEN
			eState := E_SystemState.SteamFlowing;
		END_IF

    //--------------------------------------------------------------------
    E_SystemState.SteamFlowing:     // S60: normal production
    //--------------------------------------------------------------------
		IF bEntry THEN
			tmrReadyBreak(IN := FALSE);
			tmrReadyMake(IN := FALSE);
		END_IF
	
        bControlEnable := TRUE;
		eWaterFillMode := E_WaterFillMode.RunningAutofill;
        // Ready = producing, no active faults, flow tracking setpoint
        
		tmrReadyBreak(IN := NOT _TempsInBand() OR NOT _FlowInBand(), PT := tMakeOrBreak);
		tmrReadyMake(IN := _TempsInBand() AND _FlowInBand(), PT := tMakeOrBreak);

		IF tmrReadyMake.Q THEN
			bReady := NOT stFaults.bAnyFault;
		ELSE
			bReady := FALSE;
		END_IF
		
		bDeliveryEnable := bReqDelivery AND NOT stFaults.bHmiCommLoss;
				  
        IF bReqStop THEN
            eState := E_SystemState.SesOff;
		ELSIF stFaults.bAnyFault THEN
			bReqFault := TRUE;
        END_IF

    //--------------------------------------------------------------------
    E_SystemState.Maintenance:      // S80 : manual actuation
    //--------------------------------------------------------------------
        // Outputs handled by FB_OutputHandler via HMI overrides; no auto control.
		bControlEnable := NOT stFaults.bHmiCommLoss;
		
		IF bReqExitMaint OR bReqStop THEN
			eState := E_SystemState.SesOff;
		ELSIF stFaults.bAnyFault THEN
			bReqFault := TRUE;
		END_IF

    //--------------------------------------------------------------------
    E_SystemState.Fault:            // S99 : latched fault
    //--------------------------------------------------------------------
        // All auto outputs off. Only an operator reset leaves this state,
        // and only once all latching faults have actually cleared.
        // Operator reset: clear latches, then let the monitor re-evaluate.

		IF bReqFaultReset AND NOT stFaults.bHmiCommLoss THEN
            eState := E_SystemState.InitController;
        END_IF

ELSE
    // Unknown/illegal state -> safe fallback
    eState := E_SystemState.Fault;
END_CASE

//=========================== clear serviced requests =========================
// (bReqFault is cleared at the top of the next cycle after being serviced.)
bReqStart      := FALSE;
bReqStop       := FALSE;
bReqMaint      := FALSE;
bReqExitMaint  := FALSE;
bReqFaultReset := FALSE;

METHOD PRIVATE _FlowInBand : BOOL
// check if measured flow is within tolerance of setpoint for hot start
_FlowInBand := ABS(stProcessValues.rFlowActual - stHmiSetpoints.rSetFlow) <= (GVL_SysParameters.rFlowDeadbandPct * stHmiSetpoints.rSetFlow);
END_METHOD

METHOD PRIVATE _FlowPercent : REAL
IF stProcessValues.rFlowRated > 0.0 THEN
    _FlowPercent := 100.0 * stProcessValues.rFlowActual / stProcessValues.rFlowRated;
ELSE
    _FlowPercent := 0.0;
END_IF
END_METHOD

METHOD PRIVATE _IsSpaWarm : BOOL
_IsSpaWarm := (stProcessValues.rTc1Spa >= GVL_SysParameters.rSpaWarmMinimumTemp);
END_METHOD

// TODO: real temperature bands from params (Warmup Temp V1535, Max Temp V1522).
METHOD PRIVATE _TempsInBand : BOOL
VAR
	rTempBand 	: REAL := 5.0;
	bTc1InBand	: BOOL;
	bTc2InBand	: BOOL;
	bTc3InBand	: BOOL;
END_VAR
IF (stProcessValues.rTc1Spa >= GVL_SysParameters.rSpaTempSp - rTempBand) 
	AND (stProcessValues.rTc1Spa <= GVL_SysParameters.rSpaTempSp + rTempBand) THEN
	bTc1InBand := TRUE;
END_IF

IF (stProcessValues.rTc2FlowMeter >= GVL_SysParameters.rFlowMeterTempSp - rTempBand)
    AND (stProcessValues.rTc2FlowMeter <  GVL_SysParameters.rFlowMeterTempSp + rTempBand) THEN
	bTc2InBand := TRUE;
END_IF

IF NOT bExtHeaterEnable
     OR ( (stProcessValues.rTc3External >= GVL_SysParameters.rExtMinReadyTemp)
      AND (stProcessValues.rTc3External <  GVL_SysParameters.rExtHeaterTempSp + rTempBand) ) THEN
	bTc3InBand := TRUE;
END_IF

 
 _TempsInBand := bTc1InBand AND bTc2InBand AND bTc3InBand;
END_METHOD

METHOD RequestAutofill : BOOL
VAR_INPUT
	cmd : BOOL;
END_VAR
IF cmd THEN
	bAutofillEnable := TRUE;
ELSE
	bAutofillEnable := FALSE;
END_IF
END_METHOD

METHOD RequestDelivery : BOOL
VAR_INPUT
	cmd	: BOOL;
END_VAR
IF cmd THEN 
	bReqDelivery := TRUE; 
ELSE 
	bReqDelivery := FALSE; 
END_IF
END_METHOD

METHOD RequestDpLoop : BOOL
VAR_INPUT
	cmd : BOOL;
END_VAR
IF cmd THEN 
	bDpLoopEnable := TRUE; 
ELSE 
	bDpLoopEnable := FALSE; 
END_IF
END_METHOD

METHOD RequestExitMaint : BOOL
bReqExitMaint := TRUE;
RequestExitMaint := TRUE;
END_METHOD

METHOD RequestExtHeater : BOOL
VAR_INPUT
	cmd	: BOOL;
END_VAR
IF cmd THEN
	bExtHeaterEnable := TRUE;
ELSE
	bExtHeaterEnable := FALSE;
END_IF
END_METHOD

// Force Fault. Called by MAIN when FB_FaultMonitor latches a fault.
METHOD RequestFault : BOOL
bReqFault := TRUE;
RequestFault := TRUE;
END_METHOD

// Operator reset. Only leaves Fault when latching faults have cleared.
METHOD RequestFaultReset : BOOL
bReqFaultReset := TRUE;
RequestFaultReset := TRUE;
END_METHOD

// Enter Maintenance. Honored only from SesOff.
METHOD RequestMaintenance : BOOL
bReqMaint := TRUE;
RequestMaintenance := TRUE;
END_METHOD

// SES ON. Honored only from SesOff (checked in the CASE).
METHOD RequestStart : BOOL
bReqStart := TRUE;
RequestStart := TRUE;
END_METHOD

// SES OFF / abort. Honored from any running or startup state.
METHOD RequestStop : BOOL
bReqStop := TRUE;
RequestStop := TRUE;
END_METHOD

METHOD RequestTempLoop : BOOL
VAR_INPUT
	cmd : BOOL;
END_VAR
IF cmd THEN
	bTempLoopEnable := TRUE;
ELSE
	bTempLoopEnable := FALSE;
END_IF
END_METHOD

END_FUNCTION_BLOCK

